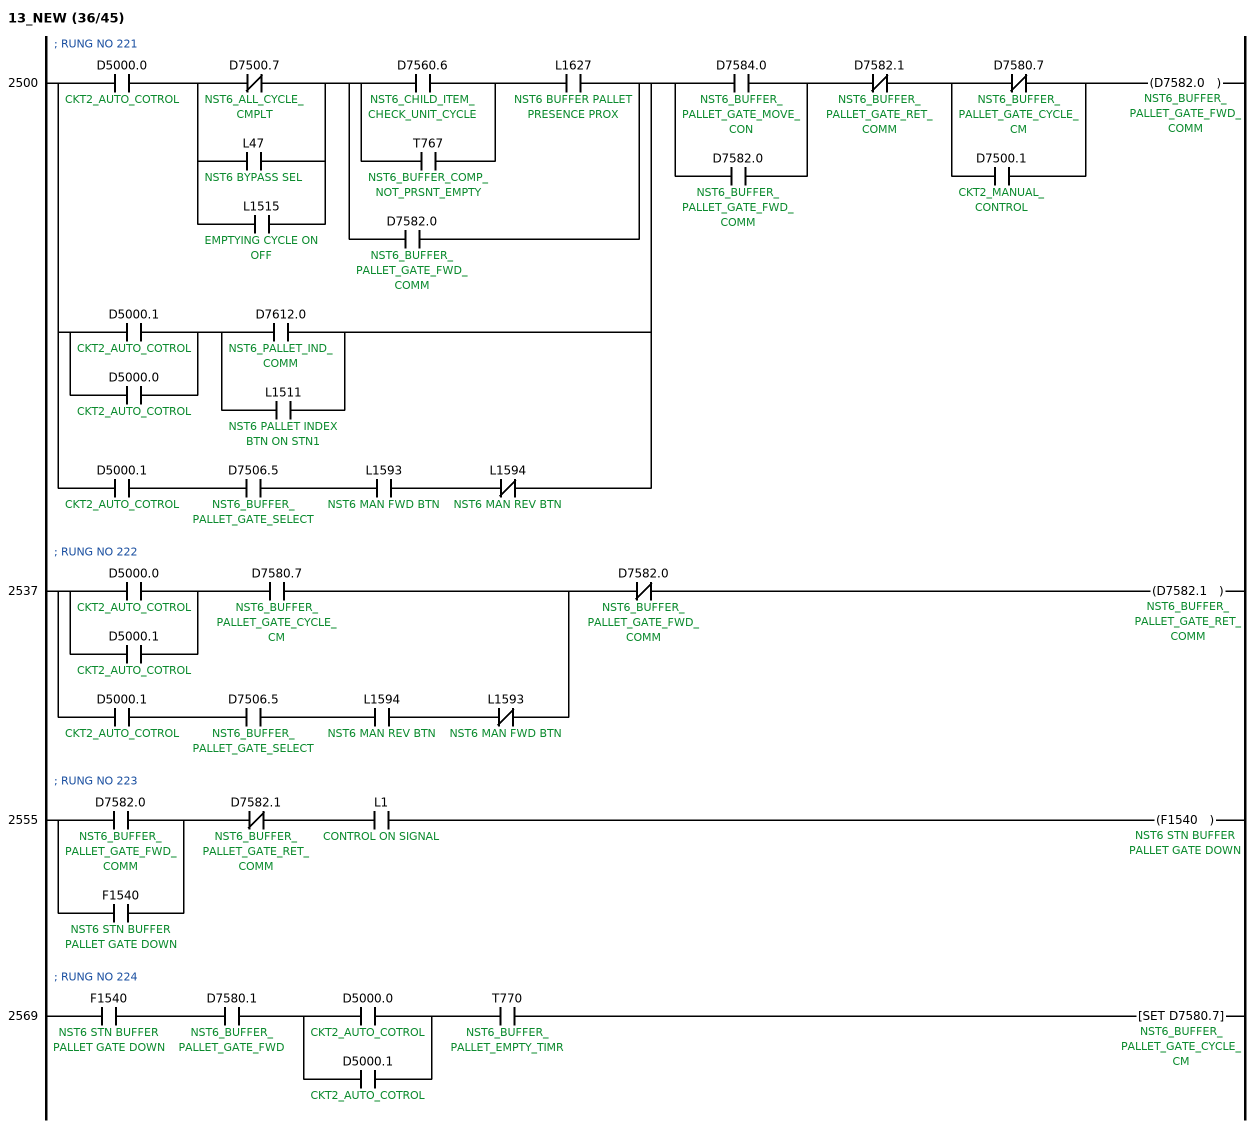
[picture p264: ladder of 13_NEW, rungs at steps 2500 to 2569]
; RUNG NO 221
2500  LD      D5000.0  ; CKT2_AUTO_COTROL
      LDI     D7500.7  ; NST6_ALL_CYCLE_CMPLT
      OR      L47  ; NST6 BYPASS SEL
      OR      L1515  ; EMPTYING CYCLE ON OFF
      ANB
      LD      D7560.6  ; NST6_CHILD_ITEM_CHECK_UNIT_CYCLE
      OR      T767  ; NST6_BUFFER_COMP_NOT_PRSNT_EMPTY
      AND     L1627  ; NST6 BUFFER PALLET PRESENCE PROX
      OR      D7582.0  ; NST6_BUFFER_PALLET_GATE_FWD_COMM
      ANB
      LD      D5000.1  ; CKT2_AUTO_COTROL
      OR      D5000.0  ; CKT2_AUTO_COTROL
      LD      D7612.0  ; NST6_PALLET_IND_COMM
      OR      L1511  ; NST6 PALLET INDEX BTN ON STN1
      ANB
      ORB
      LD      D5000.1  ; CKT2_AUTO_COTROL
      AND     D7506.5  ; NST6_BUFFER_PALLET_GATE_SELECT
      AND     L1593  ; NST6 MAN FWD BTN
      ANI     L1594  ; NST6 MAN REV BTN
      ORB
      LD      D7584.0  ; NST6_BUFFER_PALLET_GATE_MOVE_CON
      OR      D7582.0  ; NST6_BUFFER_PALLET_GATE_FWD_COMM
      ANB
      ANI     D7582.1  ; NST6_BUFFER_PALLET_GATE_RET_COMM
      LDI     D7580.7  ; NST6_BUFFER_PALLET_GATE_CYCLE_CM
      OR      D7500.1  ; CKT2_MANUAL_CONTROL
      ANB
      OUT     D7582.0  ; NST6_BUFFER_PALLET_GATE_FWD_COMM
; RUNG NO 222
2537  LD      D5000.0  ; CKT2_AUTO_COTROL
      OR      D5000.1  ; CKT2_AUTO_COTROL
      AND     D7580.7  ; NST6_BUFFER_PALLET_GATE_CYCLE_CM
      LD      D5000.1  ; CKT2_AUTO_COTROL
      AND     D7506.5  ; NST6_BUFFER_PALLET_GATE_SELECT
      AND     L1594  ; NST6 MAN REV BTN
      ANI     L1593  ; NST6 MAN FWD BTN
      ORB
      ANI     D7582.0  ; NST6_BUFFER_PALLET_GATE_FWD_COMM
      OUT     D7582.1  ; NST6_BUFFER_PALLET_GATE_RET_COMM
; RUNG NO 223
2555  LD      D7582.0  ; NST6_BUFFER_PALLET_GATE_FWD_COMM
      OR      F1540  ; NST6 STN BUFFER PALLET GATE DOWN
      ANI     D7582.1  ; NST6_BUFFER_PALLET_GATE_RET_COMM
      AND     L1  ; CONTROL ON SIGNAL
      OUT     F1540  ; NST6 STN BUFFER PALLET GATE DOWN
; RUNG NO 224
2569  LD      F1540  ; NST6 STN BUFFER PALLET GATE DOWN
      AND     D7580.1  ; NST6_BUFFER_PALLET_GATE_FWD
      LD      D5000.0  ; CKT2_AUTO_COTROL
      OR      D5000.1  ; CKT2_AUTO_COTROL
      ANB
      AND     T770  ; NST6_BUFFER_PALLET_EMPTY_TIMR
      SET     D7580.7  ; NST6_BUFFER_PALLET_GATE_CYCLE_CM
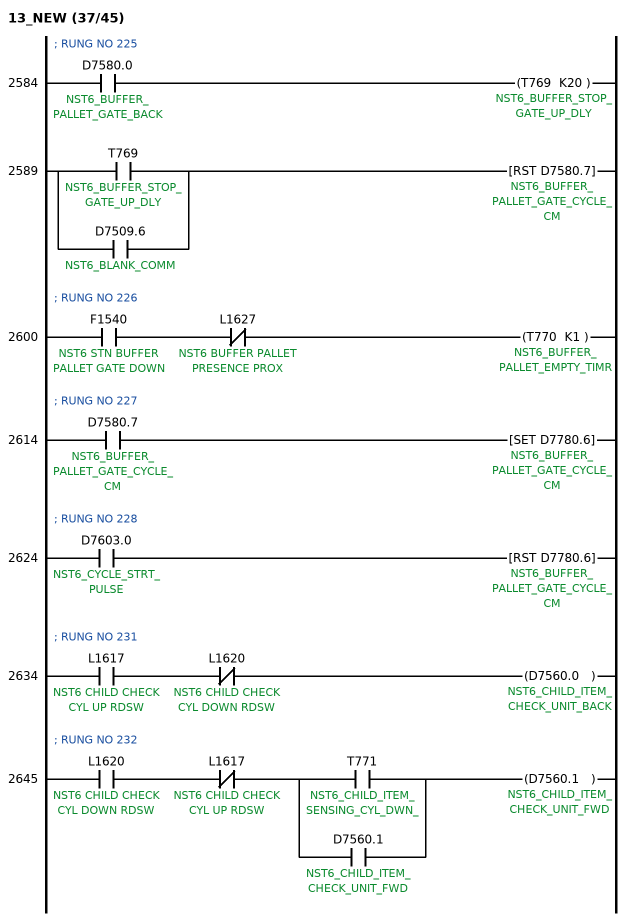
; RUNG NO 225
2584  LD      D7580.0  ; NST6_BUFFER_PALLET_GATE_BACK
      OUT     T769 K20  ; NST6_BUFFER_STOP_GATE_UP_DLY
2589  LD      T769  ; NST6_BUFFER_STOP_GATE_UP_DLY
      OR      D7509.6  ; NST6_BLANK_COMM
      RST     D7580.7  ; NST6_BUFFER_PALLET_GATE_CYCLE_CM
; RUNG NO 226
2600  LD      F1540  ; NST6 STN BUFFER PALLET GATE DOWN
      ANI     L1627  ; NST6 BUFFER PALLET PRESENCE PROX
      OUT     T770 K1  ; NST6_BUFFER_PALLET_EMPTY_TIMR
; RUNG NO 227
2614  LD      D7580.7  ; NST6_BUFFER_PALLET_GATE_CYCLE_CM
      SET     D7780.6  ; NST6_BUFFER_PALLET_GATE_CYCLE_CM
; RUNG NO 228
2624  LD      D7603.0  ; NST6_CYCLE_STRT_PULSE
      RST     D7780.6  ; NST6_BUFFER_PALLET_GATE_CYCLE_CM
; RUNG NO 231
2634  LD      L1617  ; NST6 CHILD CHECK CYL UP RDSW
      ANI     L1620  ; NST6 CHILD CHECK CYL DOWN RDSW
      OUT     D7560.0  ; NST6_CHILD_ITEM_CHECK_UNIT_BACK
; RUNG NO 232
2645  LD      L1620  ; NST6 CHILD CHECK CYL DOWN RDSW
      ANI     L1617  ; NST6 CHILD CHECK CYL UP RDSW
      LD      T771  ; NST6_CHILD_ITEM_SENSING_CYL_DWN_
      OR      D7560.1  ; NST6_CHILD_ITEM_CHECK_UNIT_FWD
      ANB
      OUT     D7560.1  ; NST6_CHILD_ITEM_CHECK_UNIT_FWD
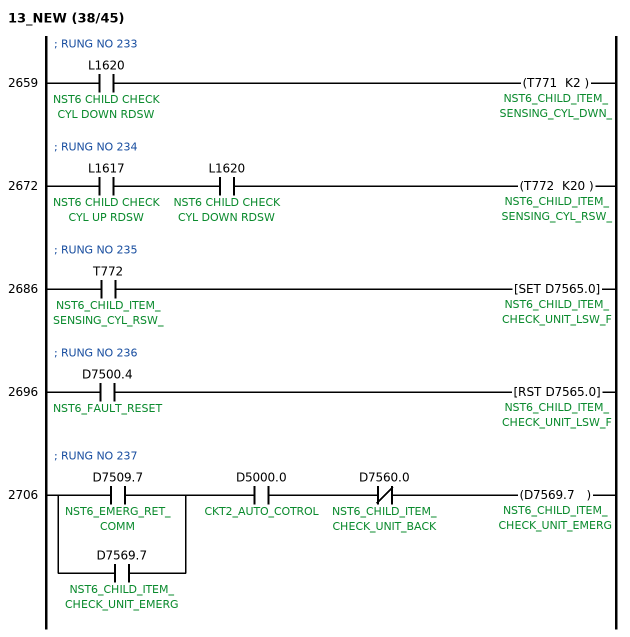
; RUNG NO 233
2659  LD      L1620  ; NST6 CHILD CHECK CYL DOWN RDSW
      OUT     T771 K2  ; NST6_CHILD_ITEM_SENSING_CYL_DWN_
; RUNG NO 234
2672  LD      L1617  ; NST6 CHILD CHECK CYL UP RDSW
      AND     L1620  ; NST6 CHILD CHECK CYL DOWN RDSW
      OUT     T772 K20  ; NST6_CHILD_ITEM_SENSING_CYL_RSW_
; RUNG NO 235
2686  LD      T772  ; NST6_CHILD_ITEM_SENSING_CYL_RSW_
      SET     D7565.0  ; NST6_CHILD_ITEM_CHECK_UNIT_LSW_F
; RUNG NO 236
2696  LD      D7500.4  ; NST6_FAULT_RESET
      RST     D7565.0  ; NST6_CHILD_ITEM_CHECK_UNIT_LSW_F
; RUNG NO 237
2706  LD      D7509.7  ; NST6_EMERG_RET_COMM
      OR      D7569.7  ; NST6_CHILD_ITEM_CHECK_UNIT_EMERG
      AND     D5000.0  ; CKT2_AUTO_COTROL
      ANI     D7560.0  ; NST6_CHILD_ITEM_CHECK_UNIT_BACK
      OUT     D7569.7  ; NST6_CHILD_ITEM_CHECK_UNIT_EMERG
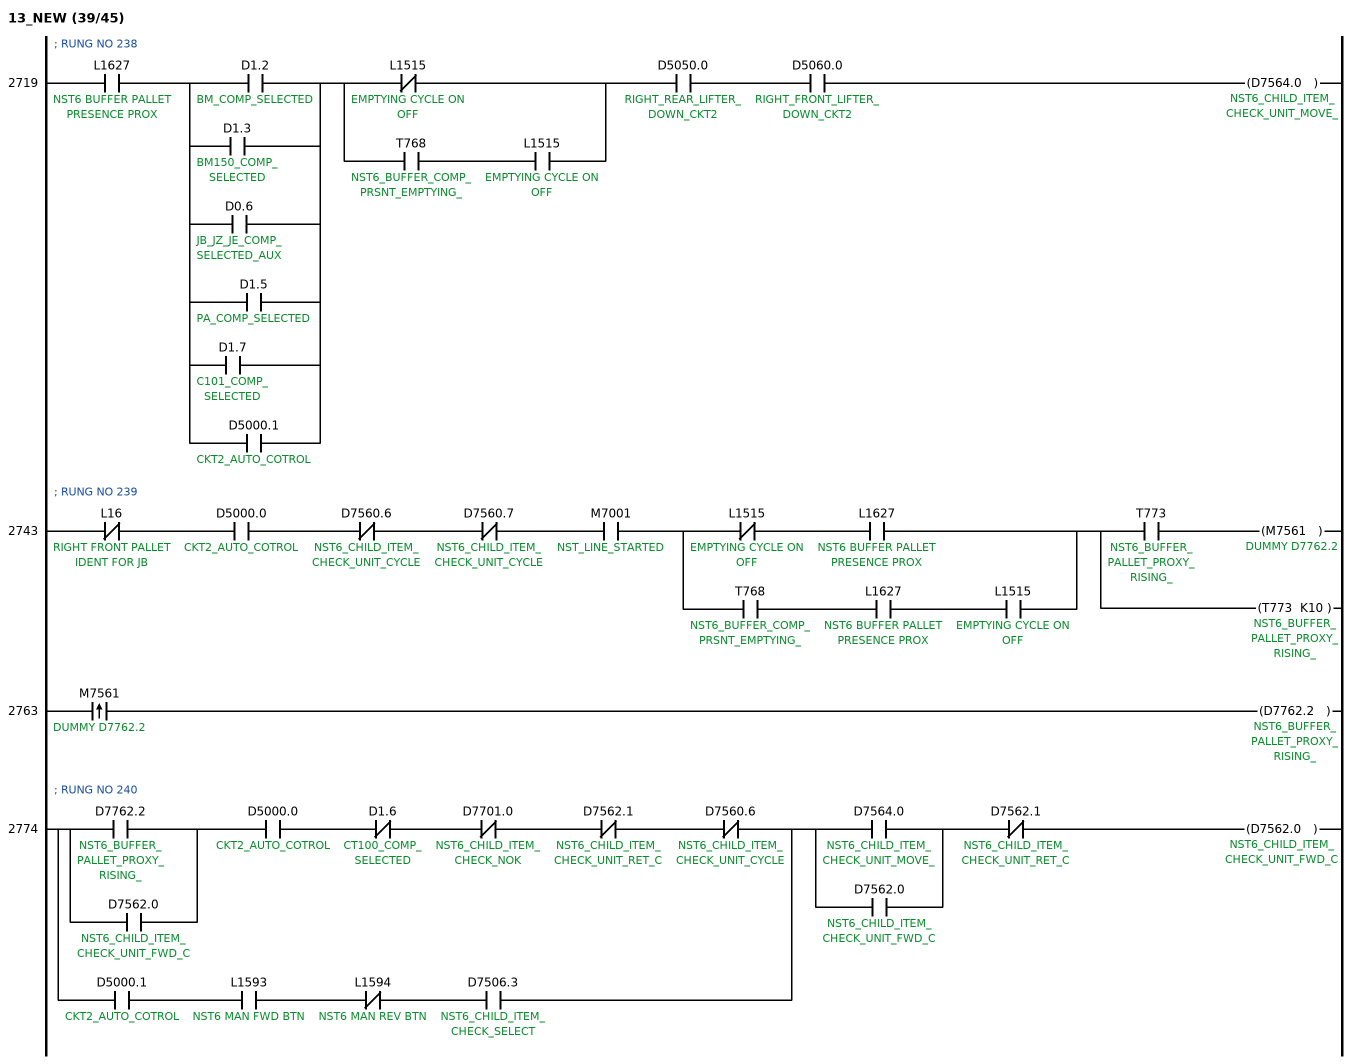
; RUNG NO 238
2719  LD      L1627  ; NST6 BUFFER PALLET PRESENCE PROX
      LD      D1.2  ; BM_COMP_SELECTED
      OR      D1.3  ; BM150_COMP_SELECTED
      OR      D0.6  ; JB_JZ_JE_COMP_SELECTED_AUX
      OR      D1.5  ; PA_COMP_SELECTED
      OR      D1.7  ; C101_COMP_SELECTED
      OR      D5000.1  ; CKT2_AUTO_COTROL
      ANB
      LDI     L1515  ; EMPTYING CYCLE ON OFF
      LD      T768  ; NST6_BUFFER_COMP_PRSNT_EMPTYING_
      AND     L1515  ; EMPTYING CYCLE ON OFF
      ORB
      ANB
      AND     D5050.0  ; RIGHT_REAR_LIFTER_DOWN_CKT2
      AND     D5060.0  ; RIGHT_FRONT_LIFTER_DOWN_CKT2
      OUT     D7564.0  ; NST6_CHILD_ITEM_CHECK_UNIT_MOVE_
; RUNG NO 239
2743  LDI     L16  ; RIGHT FRONT PALLET IDENT FOR JB
      AND     D5000.0  ; CKT2_AUTO_COTROL
      ANI     D7560.6  ; NST6_CHILD_ITEM_CHECK_UNIT_CYCLE
      ANI     D7560.7  ; NST6_CHILD_ITEM_CHECK_UNIT_CYCLE
      AND     M7001  ; NST_LINE_STARTED
      LDI     L1515  ; EMPTYING CYCLE ON OFF
      AND     L1627  ; NST6 BUFFER PALLET PRESENCE PROX
      LD      T768  ; NST6_BUFFER_COMP_PRSNT_EMPTYING_
      AND     L1627  ; NST6 BUFFER PALLET PRESENCE PROX
      AND     L1515  ; EMPTYING CYCLE ON OFF
      ORB
      ANB
      MPS
      AND     T773  ; NST6_BUFFER_PALLET_PROXY_RISING_
      OUT     M7561  ; DUMMY D7762.2
      MPP
      OUT     T773 K10  ; NST6_BUFFER_PALLET_PROXY_RISING_
2763  LDP     M7561  ; DUMMY D7762.2
      OUT     D7762.2  ; NST6_BUFFER_PALLET_PROXY_RISING_
; RUNG NO 240
2774  LD      D7762.2  ; NST6_BUFFER_PALLET_PROXY_RISING_
      OR      D7562.0  ; NST6_CHILD_ITEM_CHECK_UNIT_FWD_C
      AND     D5000.0  ; CKT2_AUTO_COTROL
      ANI     D1.6  ; CT100_COMP_SELECTED
      ANI     D7701.0  ; NST6_CHILD_ITEM_CHECK_NOK
      ANI     D7562.1  ; NST6_CHILD_ITEM_CHECK_UNIT_RET_C
      ANI     D7560.6  ; NST6_CHILD_ITEM_CHECK_UNIT_CYCLE
      LD      D5000.1  ; CKT2_AUTO_COTROL
      AND     L1593  ; NST6 MAN FWD BTN
      ANI     L1594  ; NST6 MAN REV BTN
      AND     D7506.3  ; NST6_CHILD_ITEM_CHECK_SELECT
      ORB
      LD      D7564.0  ; NST6_CHILD_ITEM_CHECK_UNIT_MOVE_
      OR      D7562.0  ; NST6_CHILD_ITEM_CHECK_UNIT_FWD_C
      ANB
      ANI     D7562.1  ; NST6_CHILD_ITEM_CHECK_UNIT_RET_C
      OUT     D7562.0  ; NST6_CHILD_ITEM_CHECK_UNIT_FWD_C
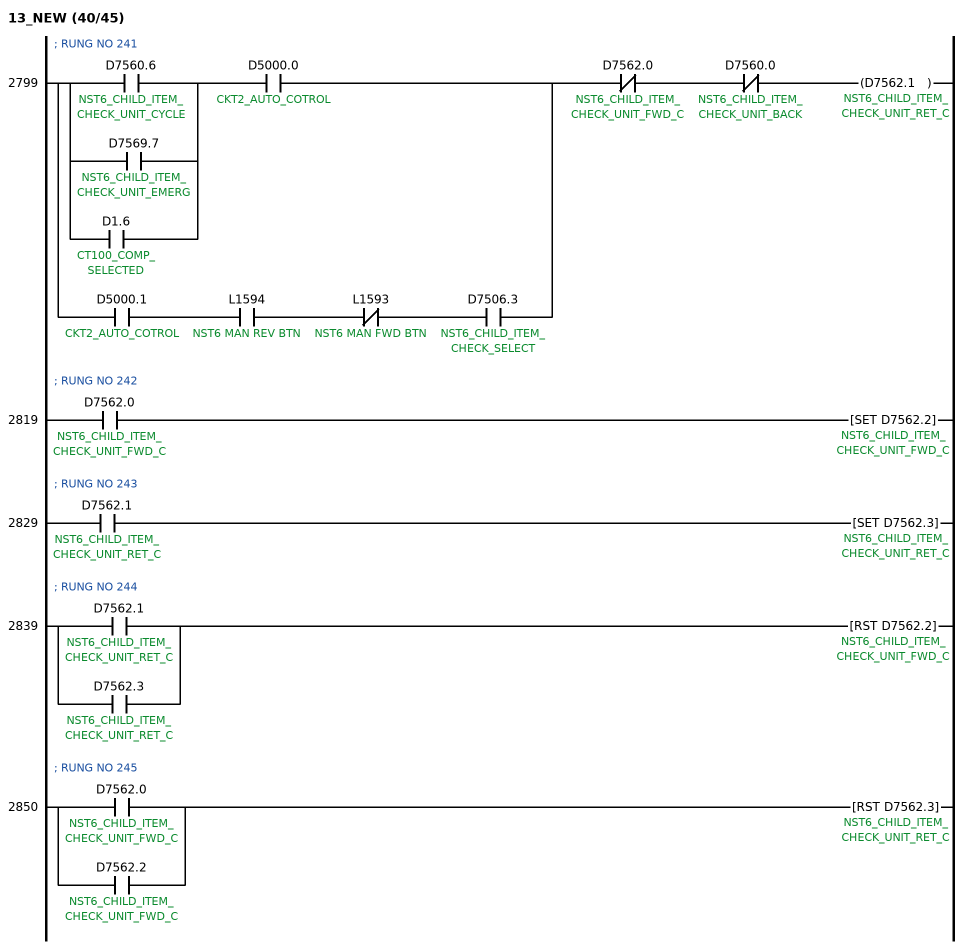
; RUNG NO 241
2799  LD      D7560.6  ; NST6_CHILD_ITEM_CHECK_UNIT_CYCLE
      OR      D7569.7  ; NST6_CHILD_ITEM_CHECK_UNIT_EMERG
      OR      D1.6  ; CT100_COMP_SELECTED
      AND     D5000.0  ; CKT2_AUTO_COTROL
      LD      D5000.1  ; CKT2_AUTO_COTROL
      AND     L1594  ; NST6 MAN REV BTN
      ANI     L1593  ; NST6 MAN FWD BTN
      AND     D7506.3  ; NST6_CHILD_ITEM_CHECK_SELECT
      ORB
      ANI     D7562.0  ; NST6_CHILD_ITEM_CHECK_UNIT_FWD_C
      ANI     D7560.0  ; NST6_CHILD_ITEM_CHECK_UNIT_BACK
      OUT     D7562.1  ; NST6_CHILD_ITEM_CHECK_UNIT_RET_C
; RUNG NO 242
2819  LD      D7562.0  ; NST6_CHILD_ITEM_CHECK_UNIT_FWD_C
      SET     D7562.2  ; NST6_CHILD_ITEM_CHECK_UNIT_FWD_C
; RUNG NO 243
2829  LD      D7562.1  ; NST6_CHILD_ITEM_CHECK_UNIT_RET_C
      SET     D7562.3  ; NST6_CHILD_ITEM_CHECK_UNIT_RET_C
; RUNG NO 244
2839  LD      D7562.1  ; NST6_CHILD_ITEM_CHECK_UNIT_RET_C
      OR      D7562.3  ; NST6_CHILD_ITEM_CHECK_UNIT_RET_C
      RST     D7562.2  ; NST6_CHILD_ITEM_CHECK_UNIT_FWD_C
; RUNG NO 245
2850  LD      D7562.0  ; NST6_CHILD_ITEM_CHECK_UNIT_FWD_C
      OR      D7562.2  ; NST6_CHILD_ITEM_CHECK_UNIT_FWD_C
      RST     D7562.3  ; NST6_CHILD_ITEM_CHECK_UNIT_RET_C
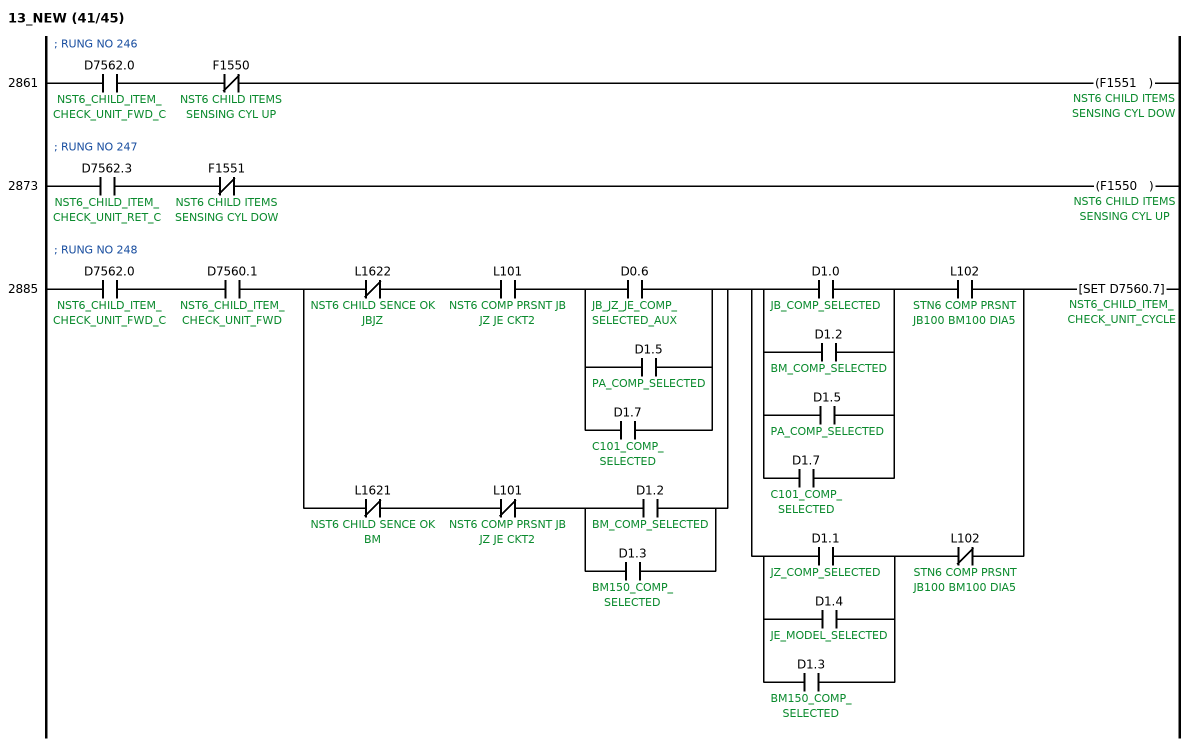
; RUNG NO 246
2861  LD      D7562.0  ; NST6_CHILD_ITEM_CHECK_UNIT_FWD_C
      ANI     F1550  ; NST6 CHILD ITEMS SENSING CYL UP
      OUT     F1551  ; NST6 CHILD ITEMS SENSING CYL DOW
; RUNG NO 247
2873  LD      D7562.3  ; NST6_CHILD_ITEM_CHECK_UNIT_RET_C
      ANI     F1551  ; NST6 CHILD ITEMS SENSING CYL DOW
      OUT     F1550  ; NST6 CHILD ITEMS SENSING CYL UP
; RUNG NO 248
2885  LD      D7562.0  ; NST6_CHILD_ITEM_CHECK_UNIT_FWD_C
      AND     D7560.1  ; NST6_CHILD_ITEM_CHECK_UNIT_FWD
      LDI     L1622  ; NST6 CHILD SENCE OK JBJZ
      AND     L101  ; NST6 COMP PRSNT JB JZ JE CKT2
      LD      D0.6  ; JB_JZ_JE_COMP_SELECTED_AUX
      OR      D1.5  ; PA_COMP_SELECTED
      OR      D1.7  ; C101_COMP_SELECTED
      ANB
      LDI     L1621  ; NST6 CHILD SENCE OK BM
      ANI     L101  ; NST6 COMP PRSNT JB JZ JE CKT2
      LD      D1.2  ; BM_COMP_SELECTED
      OR      D1.3  ; BM150_COMP_SELECTED
      ANB
      ORB
      ANB
      LD      D1.0  ; JB_COMP_SELECTED
      OR      D1.2  ; BM_COMP_SELECTED
      OR      D1.5  ; PA_COMP_SELECTED
      OR      D1.7  ; C101_COMP_SELECTED
      AND     L102  ; STN6 COMP PRSNT JB100 BM100 DIA5
      LD      D1.1  ; JZ_COMP_SELECTED
      OR      D1.4  ; JE_MODEL_SELECTED
      OR      D1.3  ; BM150_COMP_SELECTED
      ANI     L102  ; STN6 COMP PRSNT JB100 BM100 DIA5
      ORB
      ANB
      SET     D7560.7  ; NST6_CHILD_ITEM_CHECK_UNIT_CYCLE
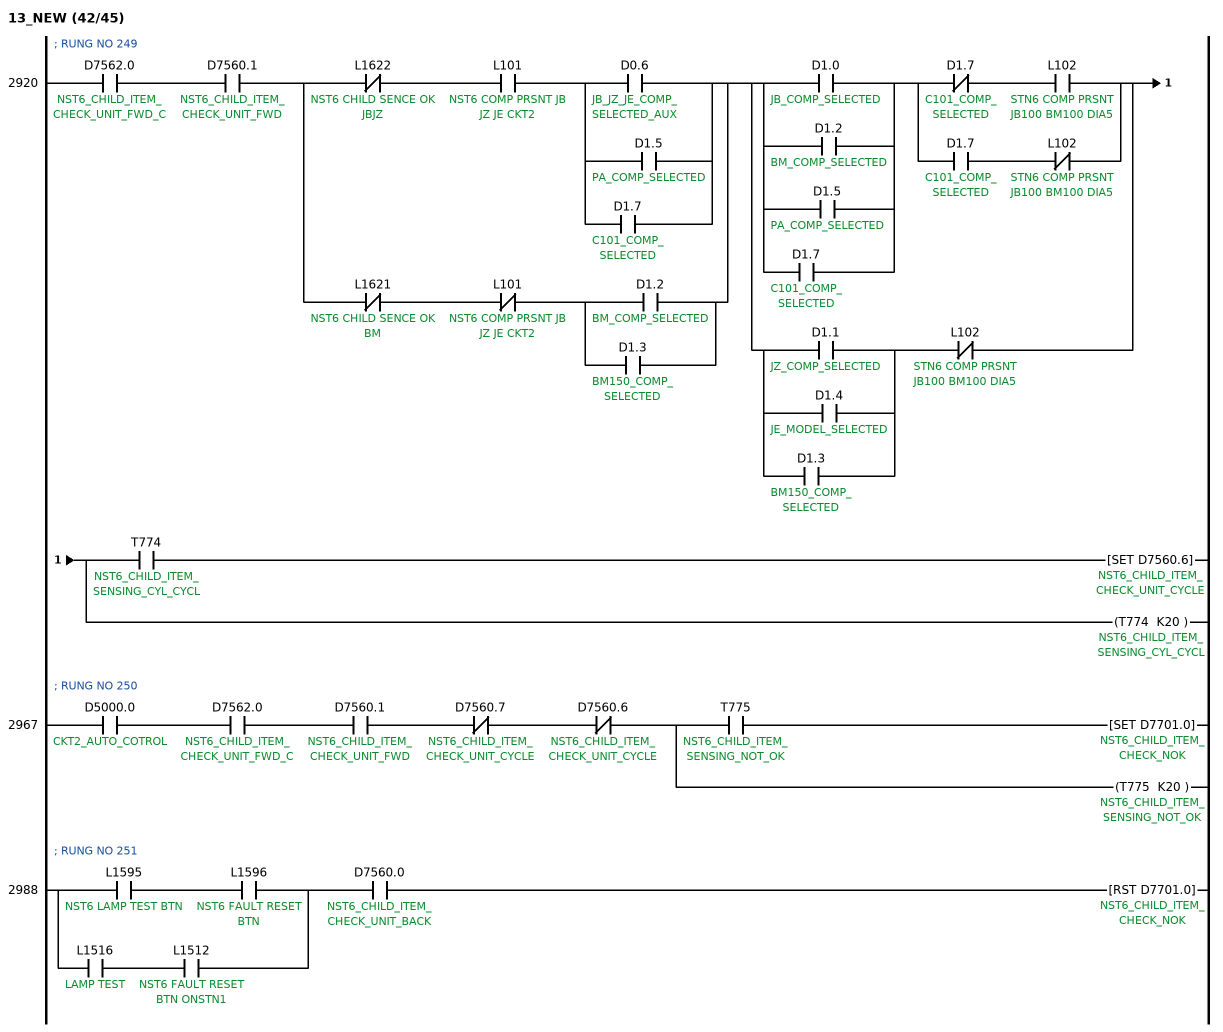
; RUNG NO 249
2920  LD      D7562.0  ; NST6_CHILD_ITEM_CHECK_UNIT_FWD_C
      AND     D7560.1  ; NST6_CHILD_ITEM_CHECK_UNIT_FWD
      LDI     L1622  ; NST6 CHILD SENCE OK JBJZ
      AND     L101  ; NST6 COMP PRSNT JB JZ JE CKT2
      LD      D0.6  ; JB_JZ_JE_COMP_SELECTED_AUX
      OR      D1.5  ; PA_COMP_SELECTED
      OR      D1.7  ; C101_COMP_SELECTED
      ANB
      LDI     L1621  ; NST6 CHILD SENCE OK BM
      ANI     L101  ; NST6 COMP PRSNT JB JZ JE CKT2
      LD      D1.2  ; BM_COMP_SELECTED
      OR      D1.3  ; BM150_COMP_SELECTED
      ANB
      ORB
      ANB
      LD      D1.0  ; JB_COMP_SELECTED
      OR      D1.2  ; BM_COMP_SELECTED
      OR      D1.5  ; PA_COMP_SELECTED
      OR      D1.7  ; C101_COMP_SELECTED
      LDI     D1.7  ; C101_COMP_SELECTED
      AND     L102  ; STN6 COMP PRSNT JB100 BM100 DIA5
      LD      D1.7  ; C101_COMP_SELECTED
      ANI     L102  ; STN6 COMP PRSNT JB100 BM100 DIA5
      ORB
      ANB
      LD      D1.1  ; JZ_COMP_SELECTED
      OR      D1.4  ; JE_MODEL_SELECTED
      OR      D1.3  ; BM150_COMP_SELECTED
      ANI     L102  ; STN6 COMP PRSNT JB100 BM100 DIA5
      ORB
      ANB
      MPS
      AND     T774  ; NST6_CHILD_ITEM_SENSING_CYL_CYCL
      SET     D7560.6  ; NST6_CHILD_ITEM_CHECK_UNIT_CYCLE
      MPP
      OUT     T774 K20  ; NST6_CHILD_ITEM_SENSING_CYL_CYCL
; RUNG NO 250
2967  LD      D5000.0  ; CKT2_AUTO_COTROL
      AND     D7562.0  ; NST6_CHILD_ITEM_CHECK_UNIT_FWD_C
      AND     D7560.1  ; NST6_CHILD_ITEM_CHECK_UNIT_FWD
      ANI     D7560.7  ; NST6_CHILD_ITEM_CHECK_UNIT_CYCLE
      ANI     D7560.6  ; NST6_CHILD_ITEM_CHECK_UNIT_CYCLE
      MPS
      AND     T775  ; NST6_CHILD_ITEM_SENSING_NOT_OK
      SET     D7701.0  ; NST6_CHILD_ITEM_CHECK_NOK
      MPP
      OUT     T775 K20  ; NST6_CHILD_ITEM_SENSING_NOT_OK
; RUNG NO 251
2988  LD      L1595  ; NST6 LAMP TEST BTN
      AND     L1596  ; NST6 FAULT RESET BTN
      LD      L1516  ; LAMP TEST
      AND     L1512  ; NST6 FAULT RESET BTN ONSTN1
      ORB
      AND     D7560.0  ; NST6_CHILD_ITEM_CHECK_UNIT_BACK
      RST     D7701.0  ; NST6_CHILD_ITEM_CHECK_NOK
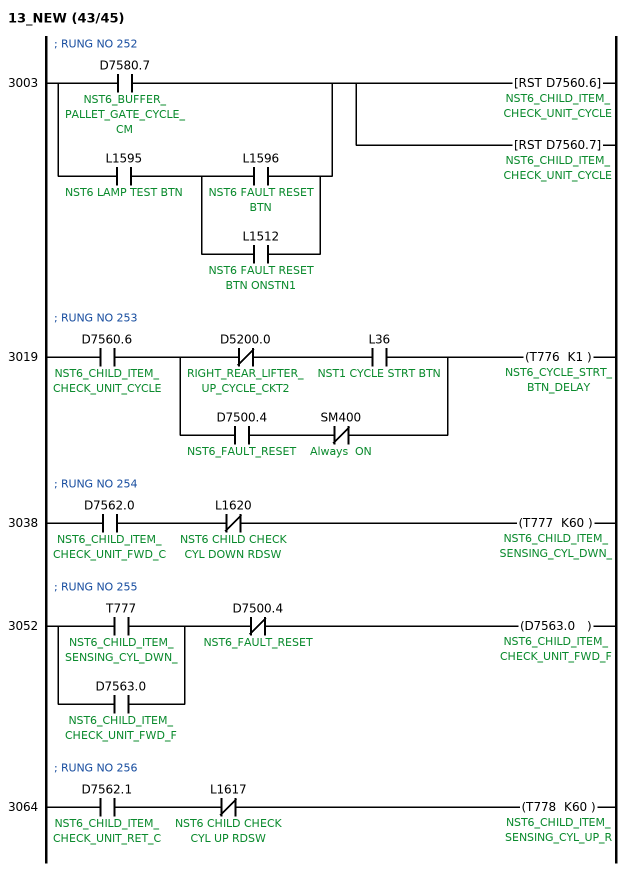
; RUNG NO 252
3003  LD      D7580.7  ; NST6_BUFFER_PALLET_GATE_CYCLE_CM
      LD      L1595  ; NST6 LAMP TEST BTN
      LD      L1596  ; NST6 FAULT RESET BTN
      OR      L1512  ; NST6 FAULT RESET BTN ONSTN1
      ANB
      ORB
      RST     D7560.6  ; NST6_CHILD_ITEM_CHECK_UNIT_CYCLE
      RST     D7560.7  ; NST6_CHILD_ITEM_CHECK_UNIT_CYCLE
; RUNG NO 253
3019  LD      D7560.6  ; NST6_CHILD_ITEM_CHECK_UNIT_CYCLE
      LDI     D5200.0  ; RIGHT_REAR_LIFTER_UP_CYCLE_CKT2
      AND     L36  ; NST1 CYCLE STRT BTN
      LD      D7500.4  ; NST6_FAULT_RESET
      ANI     SM400  ; Always  ON
      ORB
      ANB
      OUT     T776 K1  ; NST6_CYCLE_STRT_BTN_DELAY
; RUNG NO 254
3038  LD      D7562.0  ; NST6_CHILD_ITEM_CHECK_UNIT_FWD_C
      ANI     L1620  ; NST6 CHILD CHECK CYL DOWN RDSW
      OUT     T777 K60  ; NST6_CHILD_ITEM_SENSING_CYL_DWN_
; RUNG NO 255
3052  LD      T777  ; NST6_CHILD_ITEM_SENSING_CYL_DWN_
      OR      D7563.0  ; NST6_CHILD_ITEM_CHECK_UNIT_FWD_F
      ANI     D7500.4  ; NST6_FAULT_RESET
      OUT     D7563.0  ; NST6_CHILD_ITEM_CHECK_UNIT_FWD_F
; RUNG NO 256
3064  LD      D7562.1  ; NST6_CHILD_ITEM_CHECK_UNIT_RET_C
      ANI     L1617  ; NST6 CHILD CHECK CYL UP RDSW
      OUT     T778 K60  ; NST6_CHILD_ITEM_SENSING_CYL_UP_R
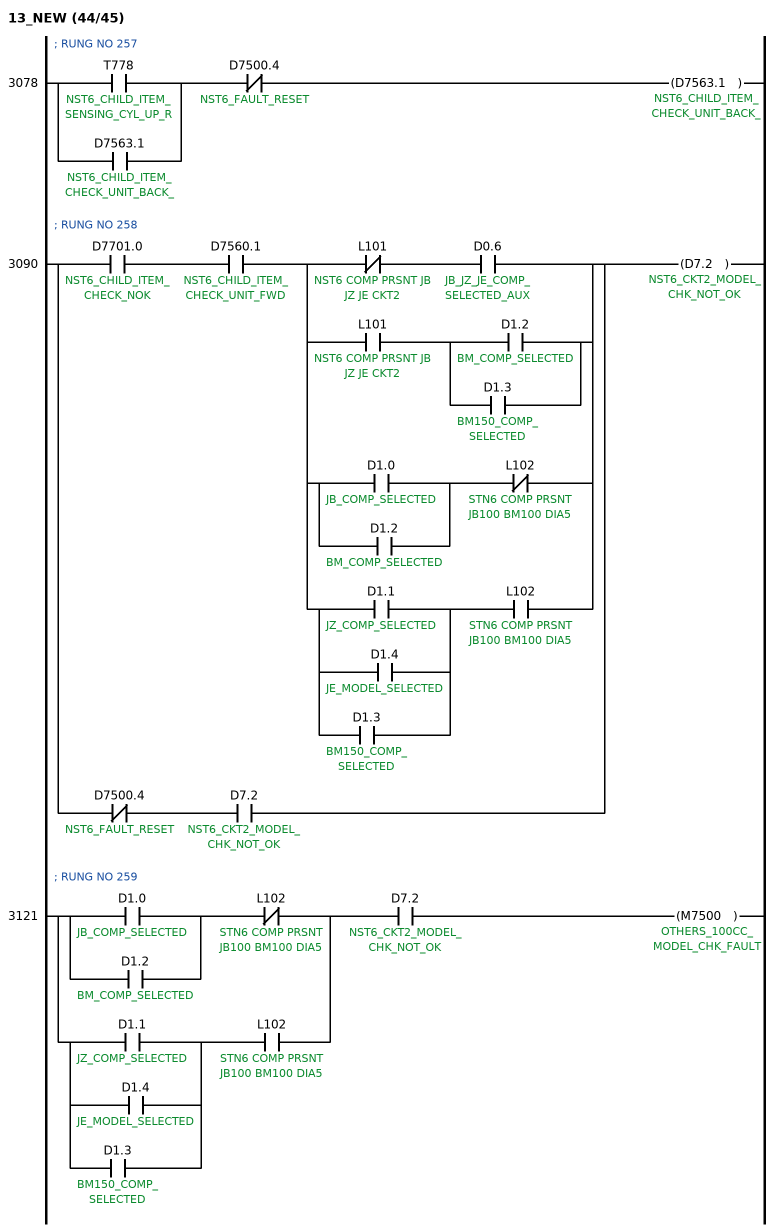
; RUNG NO 257
3078  LD      T778  ; NST6_CHILD_ITEM_SENSING_CYL_UP_R
      OR      D7563.1  ; NST6_CHILD_ITEM_CHECK_UNIT_BACK_
      ANI     D7500.4  ; NST6_FAULT_RESET
      OUT     D7563.1  ; NST6_CHILD_ITEM_CHECK_UNIT_BACK_
; RUNG NO 258
3090  LD      D7701.0  ; NST6_CHILD_ITEM_CHECK_NOK
      AND     D7560.1  ; NST6_CHILD_ITEM_CHECK_UNIT_FWD
      LDI     L101  ; NST6 COMP PRSNT JB JZ JE CKT2
      AND     D0.6  ; JB_JZ_JE_COMP_SELECTED_AUX
      LD      L101  ; NST6 COMP PRSNT JB JZ JE CKT2
      LD      D1.2  ; BM_COMP_SELECTED
      OR      D1.3  ; BM150_COMP_SELECTED
      ANB
      ORB
      LD      D1.0  ; JB_COMP_SELECTED
      OR      D1.2  ; BM_COMP_SELECTED
      ANI     L102  ; STN6 COMP PRSNT JB100 BM100 DIA5
      ORB
      LD      D1.1  ; JZ_COMP_SELECTED
      OR      D1.4  ; JE_MODEL_SELECTED
      OR      D1.3  ; BM150_COMP_SELECTED
      AND     L102  ; STN6 COMP PRSNT JB100 BM100 DIA5
      ORB
      ANB
      LDI     D7500.4  ; NST6_FAULT_RESET
      AND     D7.2  ; NST6_CKT2_MODEL_CHK_NOT_OK
      ORB
      OUT     D7.2  ; NST6_CKT2_MODEL_CHK_NOT_OK
; RUNG NO 259
3121  LD      D1.0  ; JB_COMP_SELECTED
      OR      D1.2  ; BM_COMP_SELECTED
      ANI     L102  ; STN6 COMP PRSNT JB100 BM100 DIA5
      LD      D1.1  ; JZ_COMP_SELECTED
      OR      D1.4  ; JE_MODEL_SELECTED
      OR      D1.3  ; BM150_COMP_SELECTED
      AND     L102  ; STN6 COMP PRSNT JB100 BM100 DIA5
      ORB
      AND     D7.2  ; NST6_CKT2_MODEL_CHK_NOT_OK
      OUT     M7500  ; OTHERS_100CC_MODEL_CHK_FAULT
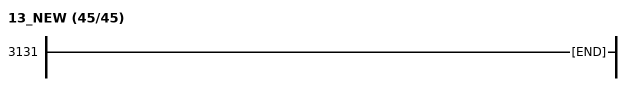
3131  END
END_PROGRAM

PROGRAM 14_OUT  // PUT NEW
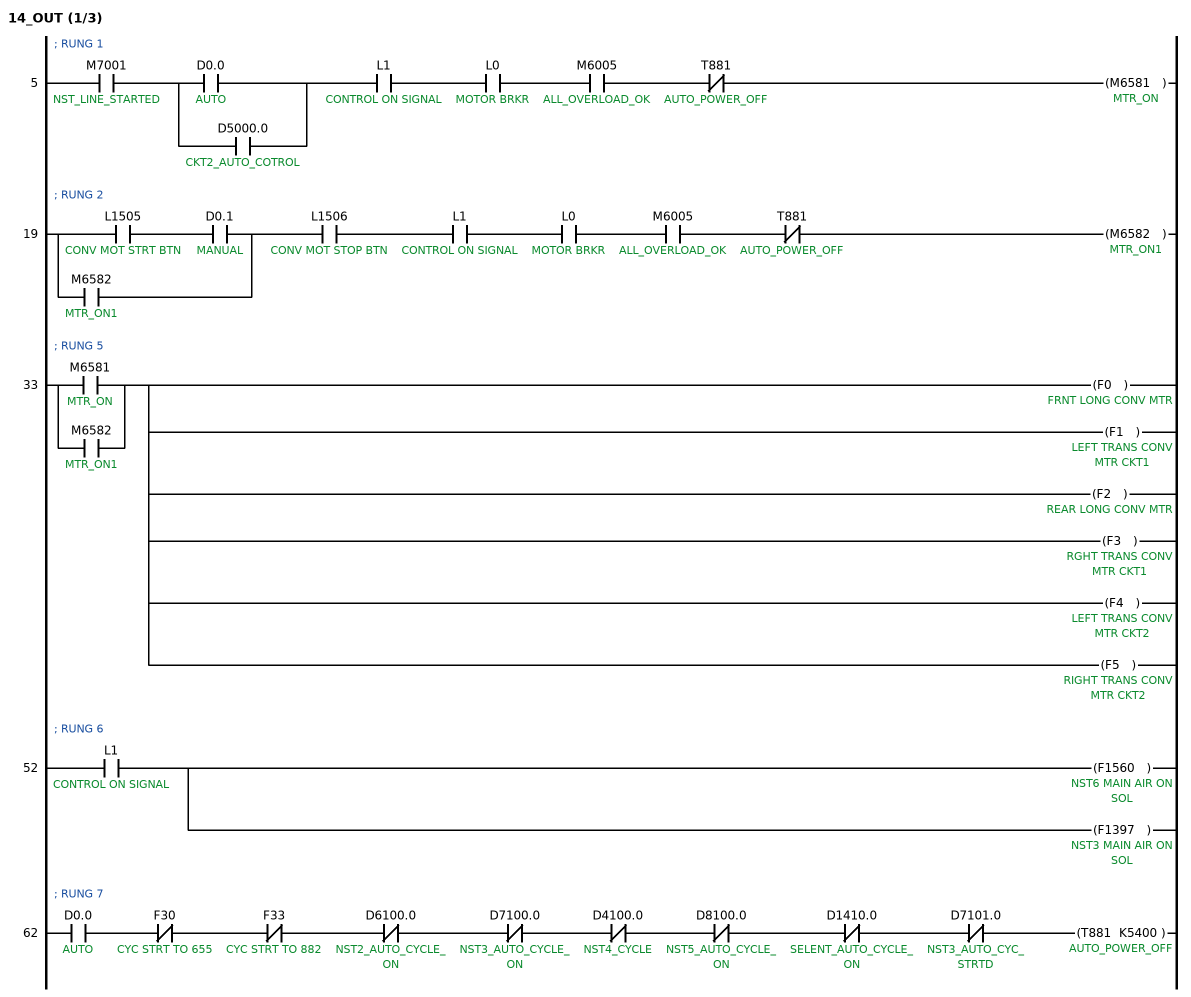
; RUNG 1
5     LD      M7001  ; NST_LINE_STARTED
      LD      D0.0  ; AUTO
      OR      D5000.0  ; CKT2_AUTO_COTROL
      ANB
      AND     L1  ; CONTROL ON SIGNAL
      AND     L0  ; MOTOR BRKR
      AND     M6005  ; ALL_OVERLOAD_OK
      ANI     T881  ; AUTO_POWER_OFF
      OUT     M6581  ; MTR_ON
; RUNG 2
19    LD      L1505  ; CONV MOT STRT BTN
      AND     D0.1  ; MANUAL
      OR      M6582  ; MTR_ON1
      AND     L1506  ; CONV MOT STOP BTN
      AND     L1  ; CONTROL ON SIGNAL
      AND     L0  ; MOTOR BRKR
      AND     M6005  ; ALL_OVERLOAD_OK
      ANI     T881  ; AUTO_POWER_OFF
      OUT     M6582  ; MTR_ON1
; RUNG 5
33    LD      M6581  ; MTR_ON
      OR      M6582  ; MTR_ON1
      OUT     F0  ; FRNT LONG CONV MTR
      OUT     F1  ; LEFT TRANS CONV MTR CKT1
      OUT     F2  ; REAR LONG CONV MTR
      OUT     F3  ; RGHT TRANS CONV MTR CKT1
      OUT     F4  ; LEFT TRANS CONV MTR CKT2
      OUT     F5  ; RIGHT TRANS CONV MTR CKT2
; RUNG 6
52    LD      L1  ; CONTROL ON SIGNAL
      OUT     F1560  ; NST6 MAIN AIR ON SOL
      OUT     F1397  ; NST3 MAIN AIR ON SOL
; RUNG 7
62    LD      D0.0  ; AUTO
      ANI     F30  ; CYC STRT TO 655
      ANI     F33  ; CYC STRT TO 882
      ANI     D6100.0  ; NST2_AUTO_CYCLE_ON
      ANI     D7100.0  ; NST3_AUTO_CYCLE_ON
      ANI     D4100.0  ; NST4_CYCLE
      ANI     D8100.0  ; NST5_AUTO_CYCLE_ON
      ANI     D1410.0  ; SELENT_AUTO_CYCLE_ON
      ANI     D7101.0  ; NST3_AUTO_CYC_STRTD
      OUT     T881 K5400  ; AUTO_POWER_OFF
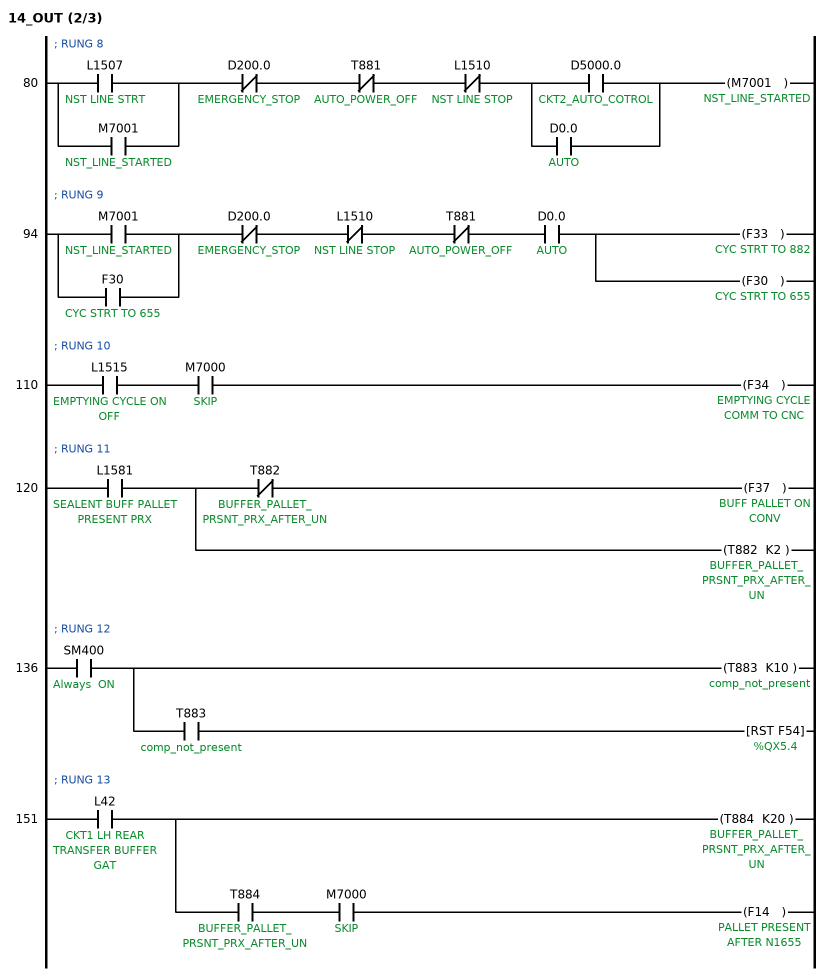
; RUNG 8
80    LD      L1507  ; NST LINE STRT
      OR      M7001  ; NST_LINE_STARTED
      ANI     D200.0  ; EMERGENCY_STOP
      ANI     T881  ; AUTO_POWER_OFF
      ANI     L1510  ; NST LINE STOP
      LD      D5000.0  ; CKT2_AUTO_COTROL
      OR      D0.0  ; AUTO
      ANB
      OUT     M7001  ; NST_LINE_STARTED
; RUNG 9
94    LD      M7001  ; NST_LINE_STARTED
      OR      F30  ; CYC STRT TO 655
      ANI     D200.0  ; EMERGENCY_STOP
      ANI     L1510  ; NST LINE STOP
      ANI     T881  ; AUTO_POWER_OFF
      AND     D0.0  ; AUTO
      OUT     F33  ; CYC STRT TO 882
      OUT     F30  ; CYC STRT TO 655
; RUNG 10
110   LD      L1515  ; EMPTYING CYCLE ON OFF
      AND     M7000  ; SKIP
      OUT     F34  ; EMPTYING CYCLE COMM TO CNC
; RUNG 11
120   LD      L1581  ; SEALENT BUFF PALLET PRESENT PRX
      MPS
      ANI     T882  ; BUFFER_PALLET_PRSNT_PRX_AFTER_UN
      OUT     F37  ; BUFF PALLET ON CONV
      MPP
      OUT     T882 K2  ; BUFFER_PALLET_PRSNT_PRX_AFTER_UN
; RUNG 12
136   LD      SM400  ; Always  ON
      OUT     T883 K10  ; comp_not_present
      AND     T883  ; comp_not_present
      RST     F54  ; %QX5.4
; RUNG 13
151   LD      L42  ; CKT1 LH REAR TRANSFER BUFFER GAT
      OUT     T884 K20  ; BUFFER_PALLET_PRSNT_PRX_AFTER_UN
      AND     T884  ; BUFFER_PALLET_PRSNT_PRX_AFTER_UN
      AND     M7000  ; SKIP
      OUT     F14  ; PALLET PRESENT AFTER N1655
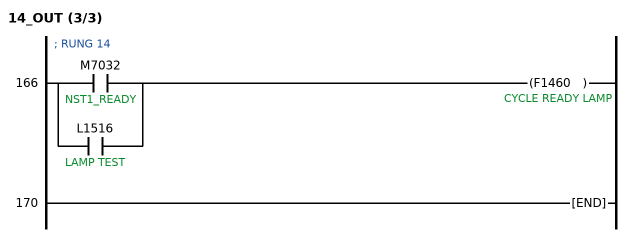
; RUNG 14
166   LD      M7032  ; NST1_READY
      OR      L1516  ; LAMP TEST
      OUT     F1460  ; CYCLE READY LAMP
170   END
END_PROGRAM

PROGRAM 15_RIGHT  // TRANSVERS CKT1
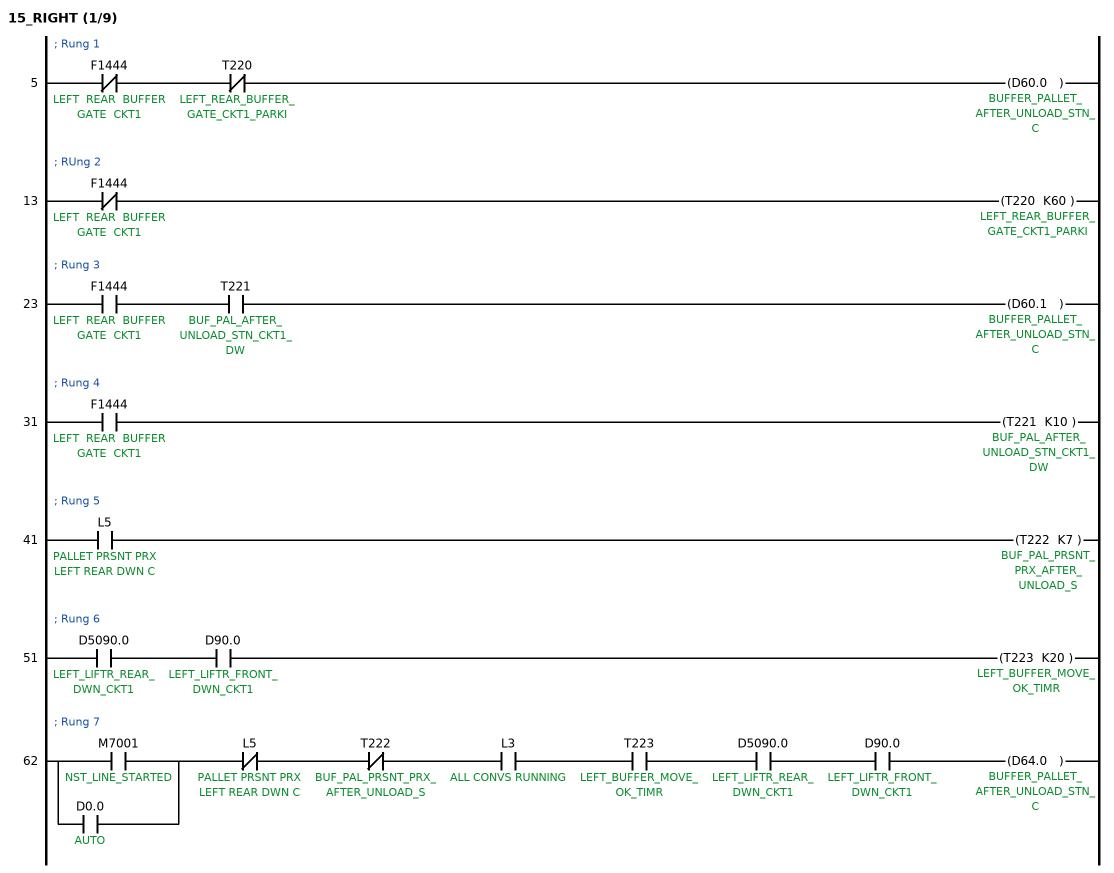
; Rung 1
5     LDI     F1444  ; LEFT  REAR  BUFFER  GATE  CKT1
      ANI     T220  ; LEFT_REAR_BUFFER_GATE_CKT1_PARKI
      OUT     D60.0  ; BUFFER_PALLET_AFTER_UNLOAD_STN_C
; RUng 2
13    LDI     F1444  ; LEFT  REAR  BUFFER  GATE  CKT1
      OUT     T220 K60  ; LEFT_REAR_BUFFER_GATE_CKT1_PARKI
; Rung 3
23    LD      F1444  ; LEFT  REAR  BUFFER  GATE  CKT1
      AND     T221  ; BUF_PAL_AFTER_UNLOAD_STN_CKT1_DW
      OUT     D60.1  ; BUFFER_PALLET_AFTER_UNLOAD_STN_C
; Rung 4
31    LD      F1444  ; LEFT  REAR  BUFFER  GATE  CKT1
      OUT     T221 K10  ; BUF_PAL_AFTER_UNLOAD_STN_CKT1_DW
; Rung 5
41    LD      L5  ; PALLET PRSNT PRX LEFT REAR DWN C
      OUT     T222 K7  ; BUF_PAL_PRSNT_PRX_AFTER_UNLOAD_S
; Rung 6
51    LD      D5090.0  ; LEFT_LIFTR_REAR_DWN_CKT1
      AND     D90.0  ; LEFT_LIFTR_FRONT_DWN_CKT1
      OUT     T223 K20  ; LEFT_BUFFER_MOVE_OK_TIMR
; Rung 7
62    LD      M7001  ; NST_LINE_STARTED
      OR      D0.0  ; AUTO
      ANI     L5  ; PALLET PRSNT PRX LEFT REAR DWN C
      ANI     T222  ; BUF_PAL_PRSNT_PRX_AFTER_UNLOAD_S
      AND     L3  ; ALL CONVS RUNNING
      AND     T223  ; LEFT_BUFFER_MOVE_OK_TIMR
      AND     D5090.0  ; LEFT_LIFTR_REAR_DWN_CKT1
      AND     D90.0  ; LEFT_LIFTR_FRONT_DWN_CKT1
      OUT     D64.0  ; BUFFER_PALLET_AFTER_UNLOAD_STN_C
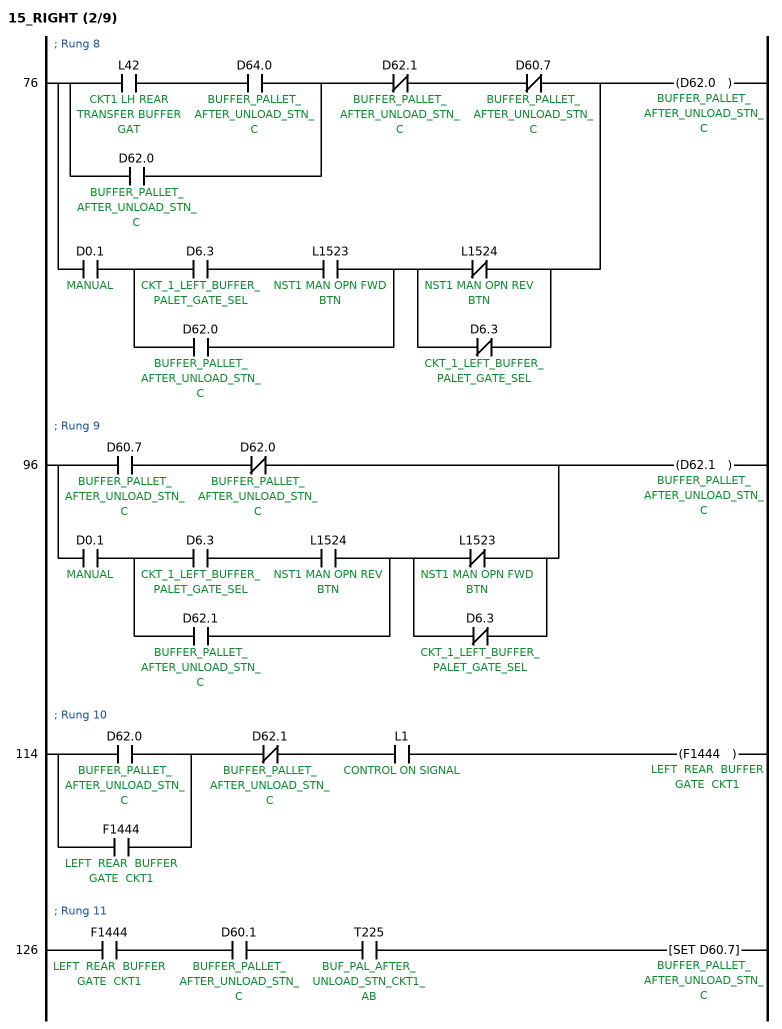
; Rung 8
76    LD      L42  ; CKT1 LH REAR TRANSFER BUFFER GAT
      AND     D64.0  ; BUFFER_PALLET_AFTER_UNLOAD_STN_C
      OR      D62.0  ; BUFFER_PALLET_AFTER_UNLOAD_STN_C
      ANI     D62.1  ; BUFFER_PALLET_AFTER_UNLOAD_STN_C
      ANI     D60.7  ; BUFFER_PALLET_AFTER_UNLOAD_STN_C
      LD      D0.1  ; MANUAL
      LD      D6.3  ; CKT_1_LEFT_BUFFER_PALET_GATE_SEL
      AND     L1523  ; NST1 MAN OPN FWD BTN
      OR      D62.0  ; BUFFER_PALLET_AFTER_UNLOAD_STN_C
      ANB
      LDI     L1524  ; NST1 MAN OPN REV BTN
      ORI     D6.3  ; CKT_1_LEFT_BUFFER_PALET_GATE_SEL
      ANB
      ORB
      OUT     D62.0  ; BUFFER_PALLET_AFTER_UNLOAD_STN_C
; Rung 9
96    LD      D60.7  ; BUFFER_PALLET_AFTER_UNLOAD_STN_C
      ANI     D62.0  ; BUFFER_PALLET_AFTER_UNLOAD_STN_C
      LD      D0.1  ; MANUAL
      LD      D6.3  ; CKT_1_LEFT_BUFFER_PALET_GATE_SEL
      AND     L1524  ; NST1 MAN OPN REV BTN
      OR      D62.1  ; BUFFER_PALLET_AFTER_UNLOAD_STN_C
      ANB
      LDI     L1523  ; NST1 MAN OPN FWD BTN
      ORI     D6.3  ; CKT_1_LEFT_BUFFER_PALET_GATE_SEL
      ANB
      ORB
      OUT     D62.1  ; BUFFER_PALLET_AFTER_UNLOAD_STN_C
; Rung 10
114   LD      D62.0  ; BUFFER_PALLET_AFTER_UNLOAD_STN_C
      OR      F1444  ; LEFT  REAR  BUFFER  GATE  CKT1
      ANI     D62.1  ; BUFFER_PALLET_AFTER_UNLOAD_STN_C
      AND     L1  ; CONTROL ON SIGNAL
      OUT     F1444  ; LEFT  REAR  BUFFER  GATE  CKT1
; Rung 11
126   LD      F1444  ; LEFT  REAR  BUFFER  GATE  CKT1
      AND     D60.1  ; BUFFER_PALLET_AFTER_UNLOAD_STN_C
      AND     T225  ; BUF_PAL_AFTER_UNLOAD_STN_CKT1_AB
      SET     D60.7  ; BUFFER_PALLET_AFTER_UNLOAD_STN_C
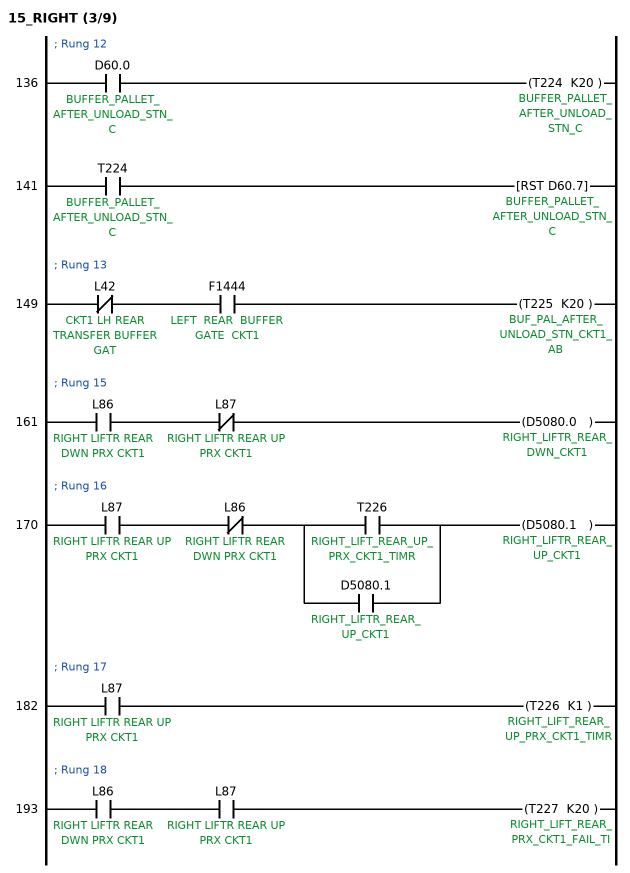
; Rung 12
136   LD      D60.0  ; BUFFER_PALLET_AFTER_UNLOAD_STN_C
      OUT     T224 K20  ; BUFFER_PALLET_AFTER_UNLOAD_STN_C
141   LD      T224  ; BUFFER_PALLET_AFTER_UNLOAD_STN_C
      RST     D60.7  ; BUFFER_PALLET_AFTER_UNLOAD_STN_C
; Rung 13
149   LDI     L42  ; CKT1 LH REAR TRANSFER BUFFER GAT
      AND     F1444  ; LEFT  REAR  BUFFER  GATE  CKT1
      OUT     T225 K20  ; BUF_PAL_AFTER_UNLOAD_STN_CKT1_AB
; Rung 15
161   LD      L86  ; RIGHT LIFTR REAR DWN PRX CKT1
      ANI     L87  ; RIGHT LIFTR REAR UP PRX CKT1
      OUT     D5080.0  ; RIGHT_LIFTR_REAR_DWN_CKT1
; Rung 16
170   LD      L87  ; RIGHT LIFTR REAR UP PRX CKT1
      ANI     L86  ; RIGHT LIFTR REAR DWN PRX CKT1
      LD      T226  ; RIGHT_LIFT_REAR_UP_PRX_CKT1_TIMR
      OR      D5080.1  ; RIGHT_LIFTR_REAR_UP_CKT1
      ANB
      OUT     D5080.1  ; RIGHT_LIFTR_REAR_UP_CKT1
; Rung 17
182   LD      L87  ; RIGHT LIFTR REAR UP PRX CKT1
      OUT     T226 K1  ; RIGHT_LIFT_REAR_UP_PRX_CKT1_TIMR
; Rung 18
193   LD      L86  ; RIGHT LIFTR REAR DWN PRX CKT1
      AND     L87  ; RIGHT LIFTR REAR UP PRX CKT1
      OUT     T227 K20  ; RIGHT_LIFT_REAR_PRX_CKT1_FAIL_TI
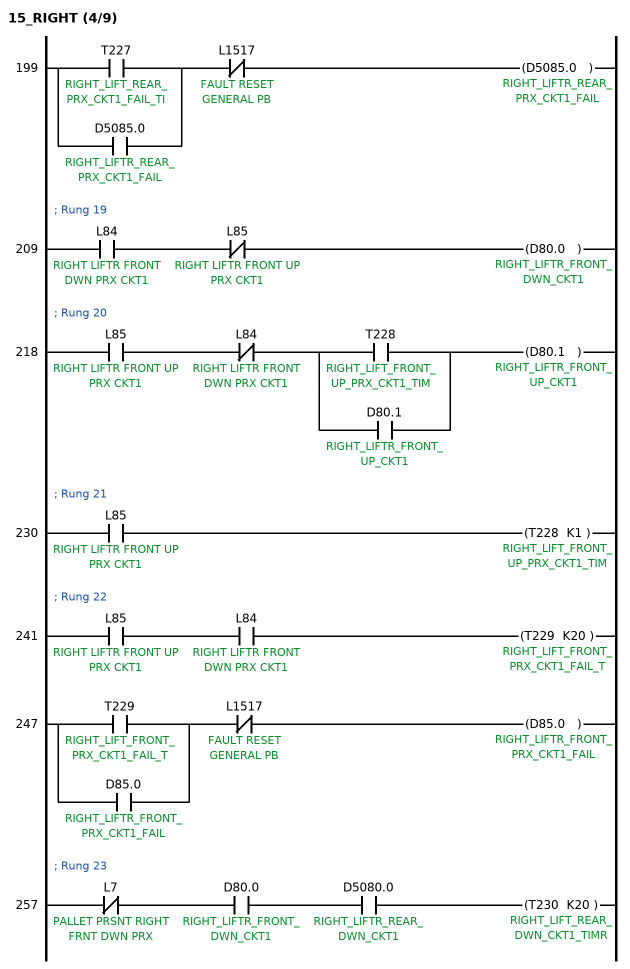
199   LD      T227  ; RIGHT_LIFT_REAR_PRX_CKT1_FAIL_TI
      OR      D5085.0  ; RIGHT_LIFTR_REAR_PRX_CKT1_FAIL
      ANI     L1517  ; FAULT RESET GENERAL PB
      OUT     D5085.0  ; RIGHT_LIFTR_REAR_PRX_CKT1_FAIL
; Rung 19
209   LD      L84  ; RIGHT LIFTR FRONT DWN PRX CKT1
      ANI     L85  ; RIGHT LIFTR FRONT UP PRX CKT1
      OUT     D80.0  ; RIGHT_LIFTR_FRONT_DWN_CKT1
; Rung 20
218   LD      L85  ; RIGHT LIFTR FRONT UP PRX CKT1
      ANI     L84  ; RIGHT LIFTR FRONT DWN PRX CKT1
      LD      T228  ; RIGHT_LIFT_FRONT_UP_PRX_CKT1_TIM
      OR      D80.1  ; RIGHT_LIFTR_FRONT_UP_CKT1
      ANB
      OUT     D80.1  ; RIGHT_LIFTR_FRONT_UP_CKT1
; Rung 21
230   LD      L85  ; RIGHT LIFTR FRONT UP PRX CKT1
      OUT     T228 K1  ; RIGHT_LIFT_FRONT_UP_PRX_CKT1_TIM
; Rung 22
241   LD      L85  ; RIGHT LIFTR FRONT UP PRX CKT1
      AND     L84  ; RIGHT LIFTR FRONT DWN PRX CKT1
      OUT     T229 K20  ; RIGHT_LIFT_FRONT_PRX_CKT1_FAIL_T
247   LD      T229  ; RIGHT_LIFT_FRONT_PRX_CKT1_FAIL_T
      OR      D85.0  ; RIGHT_LIFTR_FRONT_PRX_CKT1_FAIL
      ANI     L1517  ; FAULT RESET GENERAL PB
      OUT     D85.0  ; RIGHT_LIFTR_FRONT_PRX_CKT1_FAIL
; Rung 23
257   LDI     L7  ; PALLET PRSNT RIGHT FRNT DWN PRX
      AND     D80.0  ; RIGHT_LIFTR_FRONT_DWN_CKT1
      AND     D5080.0  ; RIGHT_LIFTR_REAR_DWN_CKT1
      OUT     T230 K20  ; RIGHT_LIFT_REAR_DWN_CKT1_TIMR
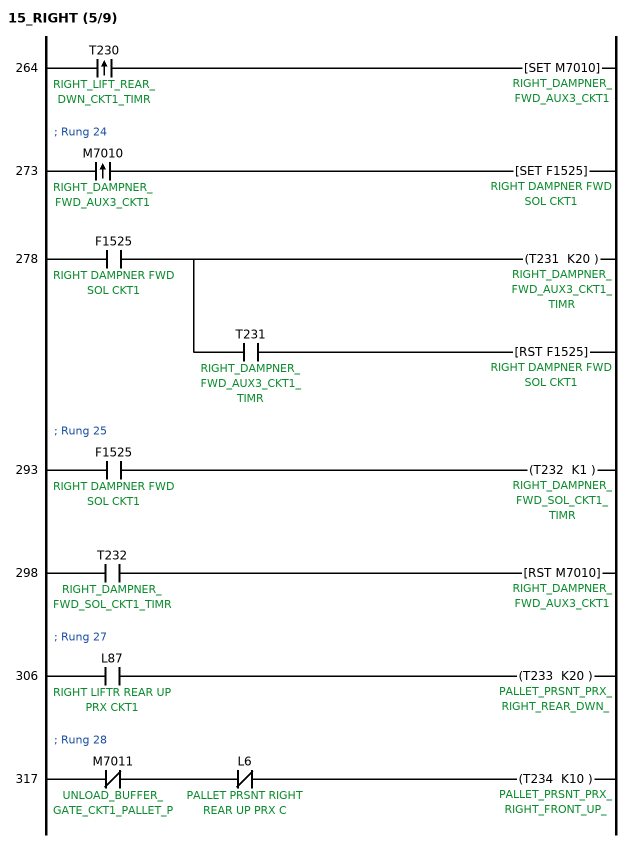
264   LDP     T230  ; RIGHT_LIFT_REAR_DWN_CKT1_TIMR
      SET     M7010  ; RIGHT_DAMPNER_FWD_AUX3_CKT1
; Rung 24
273   LDP     M7010  ; RIGHT_DAMPNER_FWD_AUX3_CKT1
      SET     F1525  ; RIGHT DAMPNER FWD SOL CKT1
278   LD      F1525  ; RIGHT DAMPNER FWD SOL CKT1
      OUT     T231 K20  ; RIGHT_DAMPNER_FWD_AUX3_CKT1_TIMR
      AND     T231  ; RIGHT_DAMPNER_FWD_AUX3_CKT1_TIMR
      RST     F1525  ; RIGHT DAMPNER FWD SOL CKT1
; Rung 25
293   LD      F1525  ; RIGHT DAMPNER FWD SOL CKT1
      OUT     T232 K1  ; RIGHT_DAMPNER_FWD_SOL_CKT1_TIMR
298   LD      T232  ; RIGHT_DAMPNER_FWD_SOL_CKT1_TIMR
      RST     M7010  ; RIGHT_DAMPNER_FWD_AUX3_CKT1
; Rung 27
306   LD      L87  ; RIGHT LIFTR REAR UP PRX CKT1
      OUT     T233 K20  ; PALLET_PRSNT_PRX_RIGHT_REAR_DWN_
; Rung 28
317   LDI     M7011  ; UNLOAD_BUFFER_GATE_CKT1_PALLET_P
      ANI     L6  ; PALLET PRSNT RIGHT REAR UP PRX C
      OUT     T234 K10  ; PALLET_PRSNT_PRX_RIGHT_FRONT_UP_
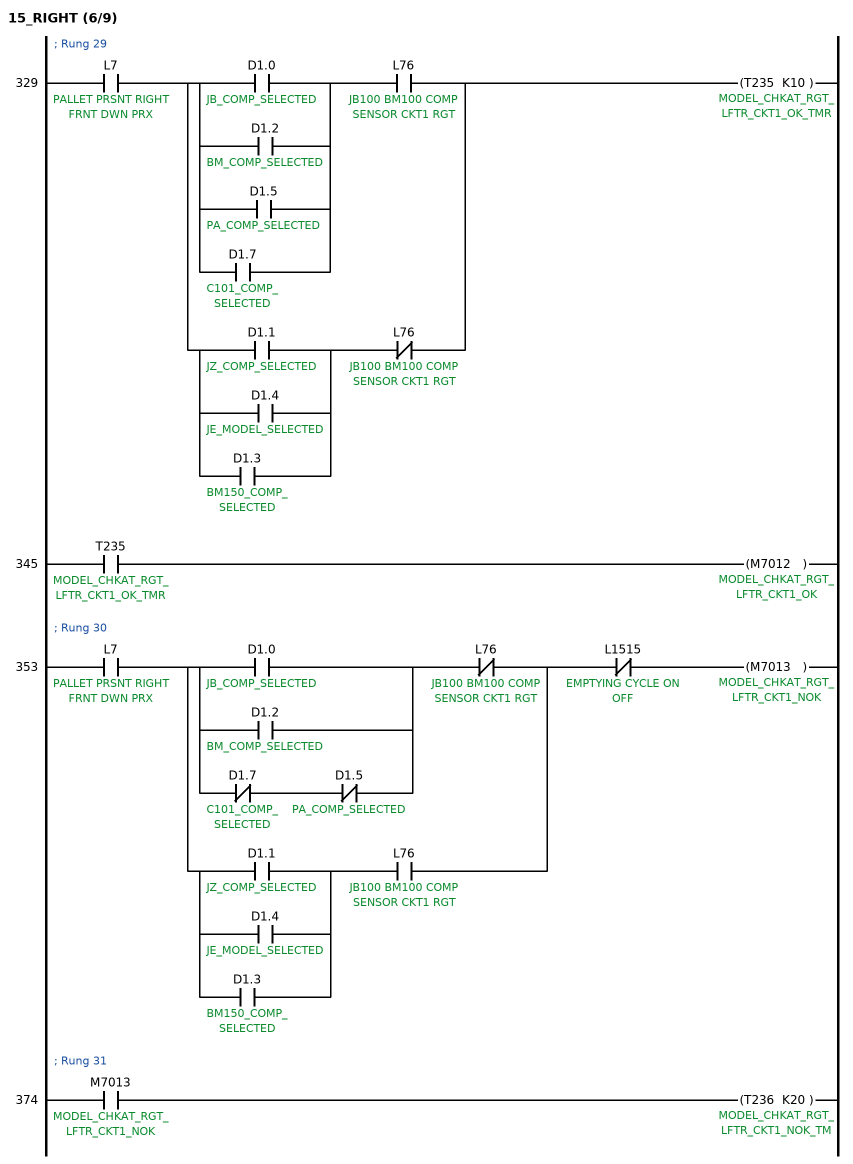
; Rung 29
329   LD      L7  ; PALLET PRSNT RIGHT FRNT DWN PRX
      LD      D1.0  ; JB_COMP_SELECTED
      OR      D1.2  ; BM_COMP_SELECTED
      OR      D1.5  ; PA_COMP_SELECTED
      OR      D1.7  ; C101_COMP_SELECTED
      AND     L76  ; JB100 BM100 COMP SENSOR CKT1 RGT
      LD      D1.1  ; JZ_COMP_SELECTED
      OR      D1.4  ; JE_MODEL_SELECTED
      OR      D1.3  ; BM150_COMP_SELECTED
      ANI     L76  ; JB100 BM100 COMP SENSOR CKT1 RGT
      ORB
      ANB
      OUT     T235 K10  ; MODEL_CHKAT_RGT_LFTR_CKT1_OK_TMR
345   LD      T235  ; MODEL_CHKAT_RGT_LFTR_CKT1_OK_TMR
      OUT     M7012  ; MODEL_CHKAT_RGT_LFTR_CKT1_OK
; Rung 30
353   LD      L7  ; PALLET PRSNT RIGHT FRNT DWN PRX
      LD      D1.0  ; JB_COMP_SELECTED
      OR      D1.2  ; BM_COMP_SELECTED
      LDI     D1.7  ; C101_COMP_SELECTED
      ANI     D1.5  ; PA_COMP_SELECTED
      ORB
      ANI     L76  ; JB100 BM100 COMP SENSOR CKT1 RGT
      LD      D1.1  ; JZ_COMP_SELECTED
      OR      D1.4  ; JE_MODEL_SELECTED
      OR      D1.3  ; BM150_COMP_SELECTED
      AND     L76  ; JB100 BM100 COMP SENSOR CKT1 RGT
      ORB
      ANB
      ANI     L1515  ; EMPTYING CYCLE ON OFF
      OUT     M7013  ; MODEL_CHKAT_RGT_LFTR_CKT1_NOK
; Rung 31
374   LD      M7013  ; MODEL_CHKAT_RGT_LFTR_CKT1_NOK
      OUT     T236 K20  ; MODEL_CHKAT_RGT_LFTR_CKT1_NOK_TM
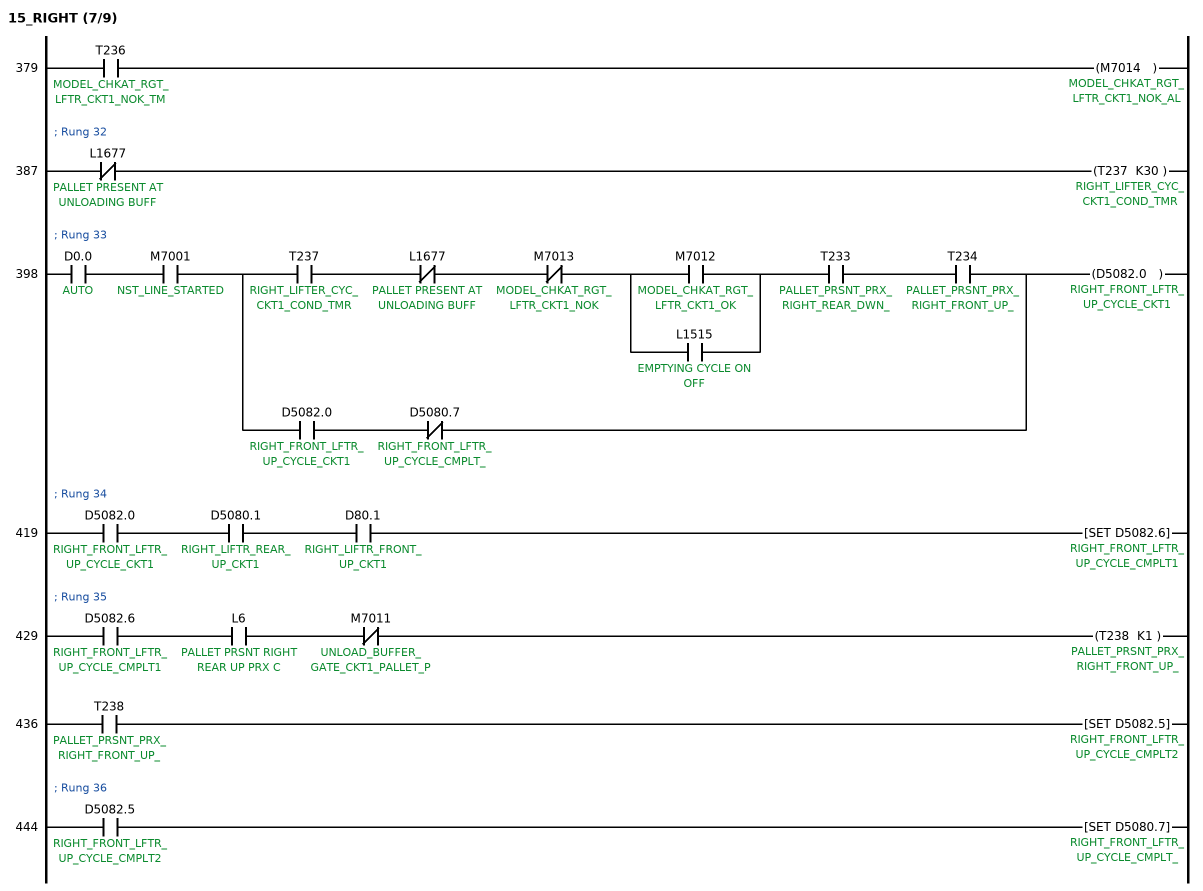
379   LD      T236  ; MODEL_CHKAT_RGT_LFTR_CKT1_NOK_TM
      OUT     M7014  ; MODEL_CHKAT_RGT_LFTR_CKT1_NOK_AL
; Rung 32
387   LDI     L1677  ; PALLET PRESENT AT UNLOADING BUFF
      OUT     T237 K30  ; RIGHT_LIFTER_CYC_CKT1_COND_TMR
; Rung 33
398   LD      D0.0  ; AUTO
      AND     M7001  ; NST_LINE_STARTED
      LD      T237  ; RIGHT_LIFTER_CYC_CKT1_COND_TMR
      ANI     L1677  ; PALLET PRESENT AT UNLOADING BUFF
      ANI     M7013  ; MODEL_CHKAT_RGT_LFTR_CKT1_NOK
      LD      M7012  ; MODEL_CHKAT_RGT_LFTR_CKT1_OK
      OR      L1515  ; EMPTYING CYCLE ON OFF
      ANB
      AND     T233  ; PALLET_PRSNT_PRX_RIGHT_REAR_DWN_
      AND     T234  ; PALLET_PRSNT_PRX_RIGHT_FRONT_UP_
      LD      D5082.0  ; RIGHT_FRONT_LFTR_UP_CYCLE_CKT1
      ANI     D5080.7  ; RIGHT_FRONT_LFTR_UP_CYCLE_CMPLT_
      ORB
      ANB
      OUT     D5082.0  ; RIGHT_FRONT_LFTR_UP_CYCLE_CKT1
; Rung 34
419   LD      D5082.0  ; RIGHT_FRONT_LFTR_UP_CYCLE_CKT1
      AND     D5080.1  ; RIGHT_LIFTR_REAR_UP_CKT1
      AND     D80.1  ; RIGHT_LIFTR_FRONT_UP_CKT1
      SET     D5082.6  ; RIGHT_FRONT_LFTR_UP_CYCLE_CMPLT1
; Rung 35
429   LD      D5082.6  ; RIGHT_FRONT_LFTR_UP_CYCLE_CMPLT1
      AND     L6  ; PALLET PRSNT RIGHT REAR UP PRX C
      ANI     M7011  ; UNLOAD_BUFFER_GATE_CKT1_PALLET_P
      OUT     T238 K1  ; PALLET_PRSNT_PRX_RIGHT_FRONT_UP_
436   LD      T238  ; PALLET_PRSNT_PRX_RIGHT_FRONT_UP_
      SET     D5082.5  ; RIGHT_FRONT_LFTR_UP_CYCLE_CMPLT2
; Rung 36
444   LD      D5082.5  ; RIGHT_FRONT_LFTR_UP_CYCLE_CMPLT2
      SET     D5080.7  ; RIGHT_FRONT_LFTR_UP_CYCLE_CMPLT_
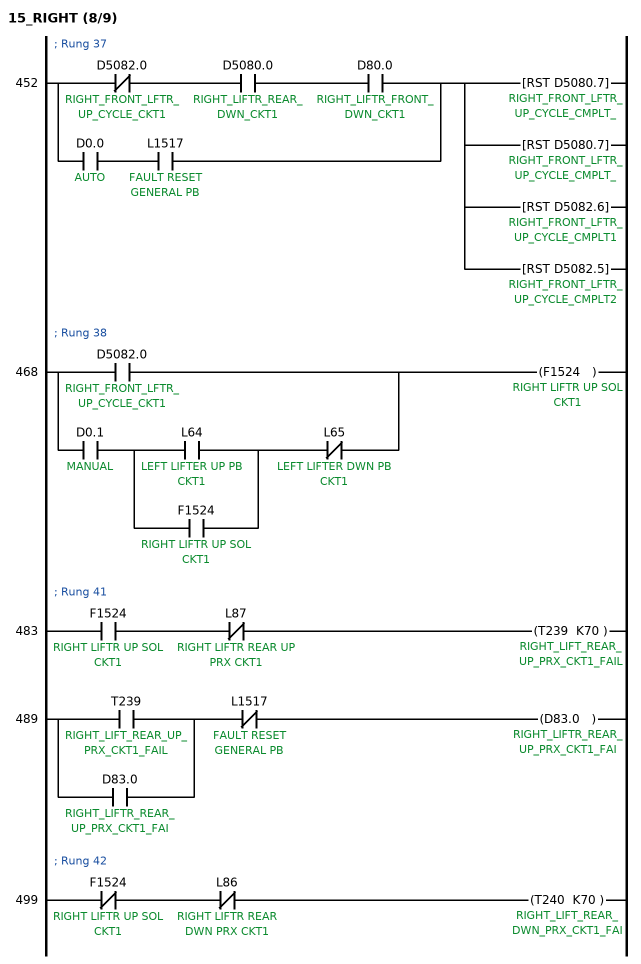
; Rung 37
452   LDI     D5082.0  ; RIGHT_FRONT_LFTR_UP_CYCLE_CKT1
      AND     D5080.0  ; RIGHT_LIFTR_REAR_DWN_CKT1
      AND     D80.0  ; RIGHT_LIFTR_FRONT_DWN_CKT1
      LD      D0.0  ; AUTO
      AND     L1517  ; FAULT RESET GENERAL PB
      ORB
      RST     D5080.7  ; RIGHT_FRONT_LFTR_UP_CYCLE_CMPLT_
      RST     D5080.7  ; RIGHT_FRONT_LFTR_UP_CYCLE_CMPLT_
      RST     D5082.6  ; RIGHT_FRONT_LFTR_UP_CYCLE_CMPLT1
      RST     D5082.5  ; RIGHT_FRONT_LFTR_UP_CYCLE_CMPLT2
; Rung 38
468   LD      D5082.0  ; RIGHT_FRONT_LFTR_UP_CYCLE_CKT1
      LD      D0.1  ; MANUAL
      LD      L64  ; LEFT LIFTER UP PB CKT1
      OR      F1524  ; RIGHT LIFTR UP SOL CKT1
      ANB
      ANI     L65  ; LEFT LIFTER DWN PB CKT1
      ORB
      OUT     F1524  ; RIGHT LIFTR UP SOL CKT1
; Rung 41
483   LD      F1524  ; RIGHT LIFTR UP SOL CKT1
      ANI     L87  ; RIGHT LIFTR REAR UP PRX CKT1
      OUT     T239 K70  ; RIGHT_LIFT_REAR_UP_PRX_CKT1_FAIL
489   LD      T239  ; RIGHT_LIFT_REAR_UP_PRX_CKT1_FAIL
      OR      D83.0  ; RIGHT_LIFTR_REAR_UP_PRX_CKT1_FAI
      ANI     L1517  ; FAULT RESET GENERAL PB
      OUT     D83.0  ; RIGHT_LIFTR_REAR_UP_PRX_CKT1_FAI
; Rung 42
499   LDI     F1524  ; RIGHT LIFTR UP SOL CKT1
      ANI     L86  ; RIGHT LIFTR REAR DWN PRX CKT1
      OUT     T240 K70  ; RIGHT_LIFT_REAR_DWN_PRX_CKT1_FAI
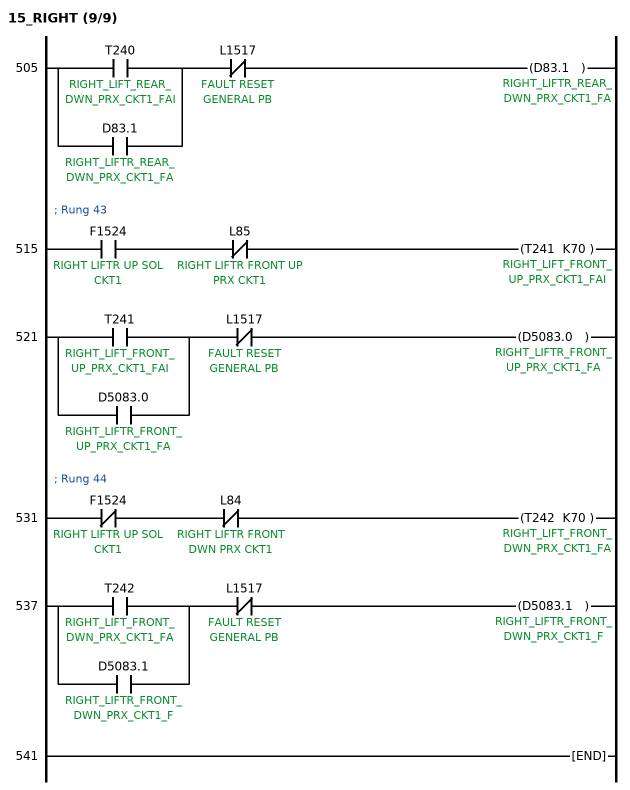
505   LD      T240  ; RIGHT_LIFT_REAR_DWN_PRX_CKT1_FAI
      OR      D83.1  ; RIGHT_LIFTR_REAR_DWN_PRX_CKT1_FA
      ANI     L1517  ; FAULT RESET GENERAL PB
      OUT     D83.1  ; RIGHT_LIFTR_REAR_DWN_PRX_CKT1_FA
; Rung 43
515   LD      F1524  ; RIGHT LIFTR UP SOL CKT1
      ANI     L85  ; RIGHT LIFTR FRONT UP PRX CKT1
      OUT     T241 K70  ; RIGHT_LIFT_FRONT_UP_PRX_CKT1_FAI
521   LD      T241  ; RIGHT_LIFT_FRONT_UP_PRX_CKT1_FAI
      OR      D5083.0  ; RIGHT_LIFTR_FRONT_UP_PRX_CKT1_FA
      ANI     L1517  ; FAULT RESET GENERAL PB
      OUT     D5083.0  ; RIGHT_LIFTR_FRONT_UP_PRX_CKT1_FA
; Rung 44
531   LDI     F1524  ; RIGHT LIFTR UP SOL CKT1
      ANI     L84  ; RIGHT LIFTR FRONT DWN PRX CKT1
      OUT     T242 K70  ; RIGHT_LIFT_FRONT_DWN_PRX_CKT1_FA
537   LD      T242  ; RIGHT_LIFT_FRONT_DWN_PRX_CKT1_FA
      OR      D5083.1  ; RIGHT_LIFTR_FRONT_DWN_PRX_CKT1_F
      ANI     L1517  ; FAULT RESET GENERAL PB
      OUT     D5083.1  ; RIGHT_LIFTR_FRONT_DWN_PRX_CKT1_F
541   END
END_PROGRAM

PROGRAM 16_SEALA  // NT APPLICATION CK1
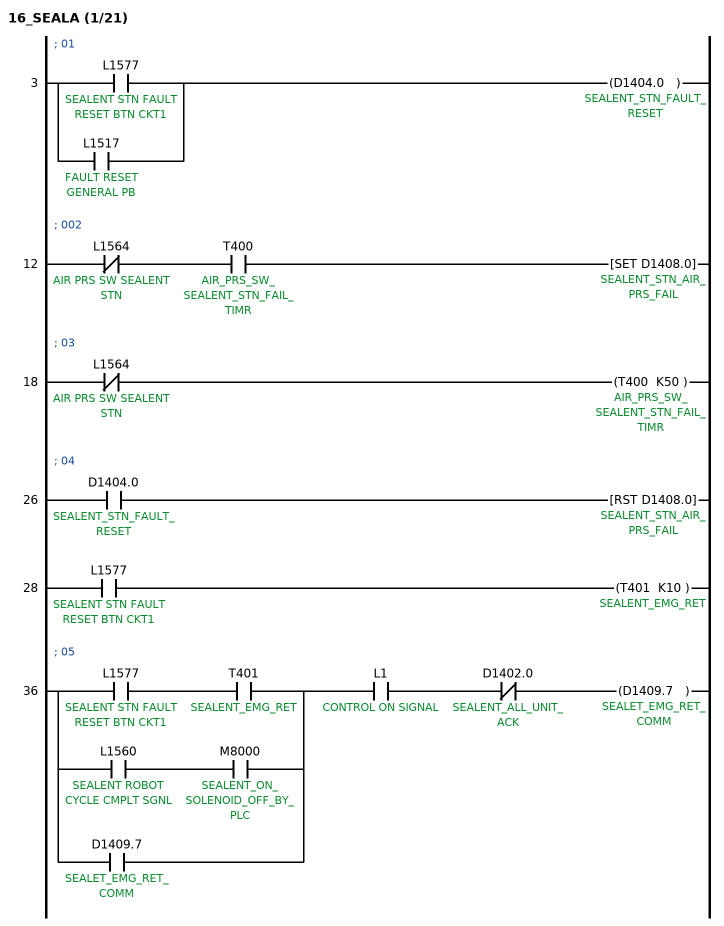
; 01
3     LD      L1577  ; SEALENT STN FAULT RESET BTN CKT1
      OR      L1517  ; FAULT RESET GENERAL PB
      OUT     D1404.0  ; SEALENT_STN_FAULT_RESET
; 
; 002
12    LDI     L1564  ; AIR PRS SW SEALENT STN
      AND     T400  ; AIR_PRS_SW_SEALENT_STN_FAIL_TIMR
      SET     D1408.0  ; SEALENT_STN_AIR_PRS_FAIL
; 03
18    LDI     L1564  ; AIR PRS SW SEALENT STN
      OUT     T400 K50  ; AIR_PRS_SW_SEALENT_STN_FAIL_TIMR
; 04
26    LD      D1404.0  ; SEALENT_STN_FAULT_RESET
      RST     D1408.0  ; SEALENT_STN_AIR_PRS_FAIL
28    LD      L1577  ; SEALENT STN FAULT RESET BTN CKT1
      OUT     T401 K10  ; SEALENT_EMG_RET
; 05
36    LD      L1577  ; SEALENT STN FAULT RESET BTN CKT1
      AND     T401  ; SEALENT_EMG_RET
      LD      L1560  ; SEALENT ROBOT CYCLE CMPLT SGNL
      AND     M8000  ; SEALENT_ON_SOLENOID_OFF_BY_PLC
      ORB
      OR      D1409.7  ; SEALET_EMG_RET_COMM
      AND     L1  ; CONTROL ON SIGNAL
      ANI     D1402.0  ; SEALENT_ALL_UNIT_ACK
      OUT     D1409.7  ; SEALET_EMG_RET_COMM
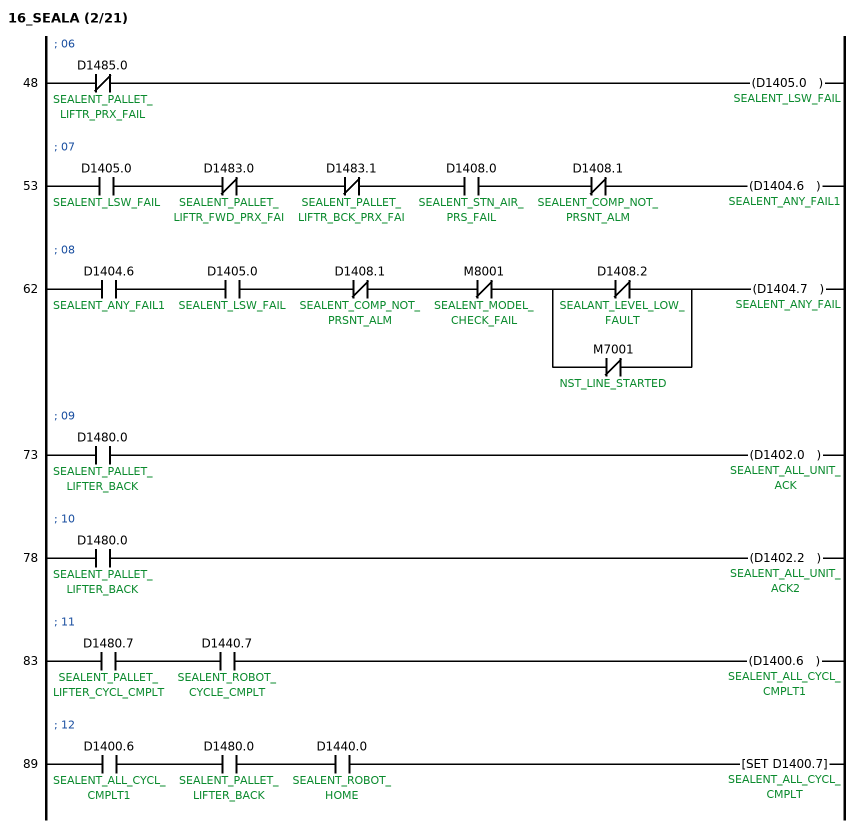
; 06
48    LDI     D1485.0  ; SEALENT_PALLET_LIFTR_PRX_FAIL
      OUT     D1405.0  ; SEALENT_LSW_FAIL
; 07
53    LD      D1405.0  ; SEALENT_LSW_FAIL
      ANI     D1483.0  ; SEALENT_PALLET_LIFTR_FWD_PRX_FAI
      ANI     D1483.1  ; SEALENT_PALLET_LIFTR_BCK_PRX_FAI
      AND     D1408.0  ; SEALENT_STN_AIR_PRS_FAIL
      ANI     D1408.1  ; SEALENT_COMP_NOT_PRSNT_ALM
      OUT     D1404.6  ; SEALENT_ANY_FAIL1
; 08
62    LD      D1404.6  ; SEALENT_ANY_FAIL1
      AND     D1405.0  ; SEALENT_LSW_FAIL
      ANI     D1408.1  ; SEALENT_COMP_NOT_PRSNT_ALM
      ANI     M8001  ; SEALENT_MODEL_CHECK_FAIL
      LDI     D1408.2  ; SEALANT_LEVEL_LOW_FAULT
      ORI     M7001  ; NST_LINE_STARTED
      ANB
      OUT     D1404.7  ; SEALENT_ANY_FAIL
; 09
73    LD      D1480.0  ; SEALENT_PALLET_LIFTER_BACK
      OUT     D1402.0  ; SEALENT_ALL_UNIT_ACK
; 10
78    LD      D1480.0  ; SEALENT_PALLET_LIFTER_BACK
      OUT     D1402.2  ; SEALENT_ALL_UNIT_ACK2
; 11
83    LD      D1480.7  ; SEALENT_PALLET_LIFTER_CYCL_CMPLT
      AND     D1440.7  ; SEALENT_ROBOT_CYCLE_CMPLT
      OUT     D1400.6  ; SEALENT_ALL_CYCL_CMPLT1
; 12
89    LD      D1400.6  ; SEALENT_ALL_CYCL_CMPLT1
      AND     D1480.0  ; SEALENT_PALLET_LIFTER_BACK
      AND     D1440.0  ; SEALENT_ROBOT_HOME
      SET     D1400.7  ; SEALENT_ALL_CYCL_CMPLT
